KUKA KRL program: MyProgram_115().src

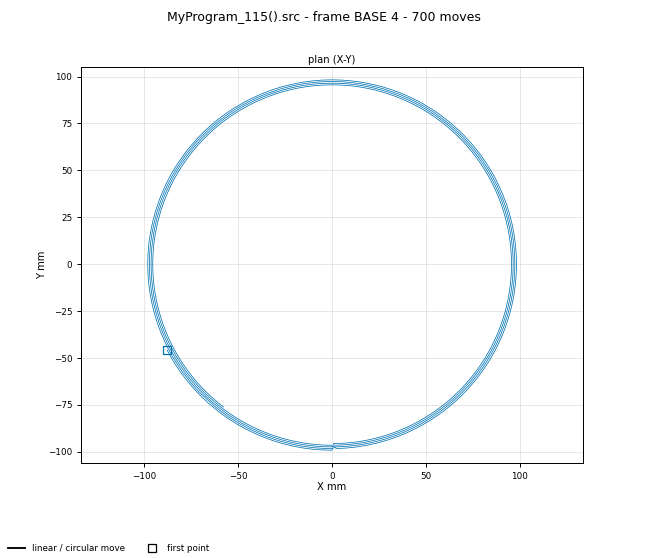
[picture p0: tool path of MyProgram_115().src in frame BASE 4, 700 of 700 moves have a stored position in this frame; points joined in program order, loops and branches not executed]
&ACCESS RVP
&REL 1
&PARAM TEMPLATE = C:\KRC\Roboter\Template\vorgabe
&PARAM EDITMASK = *
DEF MyProgram_115()
; ---- Setting reference (Base) ----
$BASE = BASE_DATA[4]

; --------------------------
; ---- Setting tool (TCP) ----
$TOOL = TOOL_DATA[3]
; --------------------------

$VEL.CP = VEL_APROX_PRINT
Startdeposition()
$VEL.CP = VEL_PRINT
LIN {X -87.9796,Y -45.6346,Z 99,A -156.4793,B 24.9343,C -1.8721,E1 24.8586,E2 241.8644} C_DIS
LIN {X -86.3816,Y -48.5897,Z 99,A -154.8089,B 24.9353,C -1.8576,E1 24.8608,E2 240.2197} C_DIS
LIN {X -84.702,Y -51.4607,Z 99,A -152.4572,B 24.9346,C -1.8672,E1 24.8642,E2 237.8331} C_DIS
LIN {X -82.3707,Y -55.1181,Z 99,A -150.0558,B 24.9354,C -1.8571,E1 24.8679,E2 235.4438} C_DIS
LIN {X -80.7403,Y -57.4774,Z 99,A -147.4324,B 24.9333,C -1.8865,E1 24.8723,E2 232.7375} C_DIS
LIN {X -77.3944,Y -61.9119,Z 99,A -145.2941,B 24.9364,C -1.8414,E1 24.8758,E2 230.6966} C_DIS
LIN {X -72.9328,Y -67.1078,Z 99,A -141.2258,B 24.9368,C -1.8361,E1 24.8833,E2 226.6225} C_DIS
LIN {X -70.3897,Y -69.7707,Z 99,A -138.1583,B 24.9348,C -1.8645,E1 24.8895,E2 223.4743} C_DIS
LIN {X -66.5722,Y -73.4243,Z 99,A -135.9548,B 24.9373,C -1.8283,E1 24.8938,E2 221.3481} C_DIS
LIN {X -64.5573,Y -75.2007,Z 99,A -133.5935,B 24.9356,C -1.8539,E1 24.899,E2 218.9168} C_DIS
LIN {X -60.7037,Y -78.3439,Z 99,A -131.5906,B 24.9381,C -1.8177,E1 24.9032,E2 216.9924} C_DIS
LIN {X -57.0304,Y -81.0586,Z 99,A -129.0585,B 24.9386,C -1.8094,E1 24.9089,E2 214.4714} C_DIS
LIN {X -53.8485,Y -83.2053,Z 99,A -126.6505,B 24.9384,C -1.8125,E1 24.9145,E2 212.0479} C_DIS
LIN {X -50.892,Y -85.0464,Z 99,A -124.5261,B 24.9384,C -1.8135,E1 24.9196,E2 209.9146} C_DIS
LIN {X -47.2587,Y -87.1163,Z 99,A -122.248,B 24.9389,C -1.8053,E1 24.9252,E2 207.6496} C_DIS
LIN {X -44.1537,Y -88.7306,Z 99,A -120.2492,B 24.9391,C -1.8018,E1 24.9301,E2 205.6535} C_DIS
LIN {X -40.0948,Y -90.6385,Z 99,A -117.5727,B 24.9391,C -1.8018,E1 24.9369,E2 202.9703} C_DIS
LIN {X -36.8273,Y -92.0148,Z 99,A -115.7096,B 24.9397,C -1.7931,E1 24.9417,E2 201.1239} C_DIS
LIN {X -32.0757,Y -93.7762,Z 99,A -112.6664,B 24.9397,C -1.7946,E1 24.9497,E2 198.0711} C_DIS
LIN {X -29.2016,Y -94.7097,Z 99,A -111.0211,B 24.94,C -1.7896,E1 24.9541,E2 196.4347} C_DIS
LIN {X -26.1849,Y -95.5883,Z 99,A -108.5473,B 24.9384,C -1.8125,E1 24.9609,E2 193.9027} C_DIS
LIN {X -22.6221,Y -96.4935,Z 99,A -106.9162,B 24.9397,C -1.7932,E1 24.9652,E2 192.3152} C_DIS
LIN {X -18.9638,Y -97.2783,Z 99,A -104.6871,B 24.9397,C -1.7947,E1 24.9713,E2 190.0799} C_DIS
LIN {X -15.5993,Y -97.875,Z 99,A -102.0723,B 24.9381,C -1.8179,E1 24.9787,E2 187.4077} C_DIS
LIN {X -11.2084,Y -98.4739,Z 99,A -100.3885,B 24.9403,C -1.7848,E1 24.9832,E2 185.8012} C_DIS
LIN {X -7.2101,Y -98.847,Z 99,A -97.791,B 24.9396,C -1.7949,E1 24.9904,E2 183.1785} C_DIS
LIN {X -0.3589,Y -99.1089,Z 99,A -93.8886,B 24.9397,C -1.7932,E1 25.0013,E2 179.2797} C_DIS
LIN {X -0.3589,Y -99.1089,Z 99,A -93.8886,B 24.9397,C -1.7932,E1 25.0013,E2 179.2797} C_DIS
Enddeposition()
LIN {X 0.6693,Y -98.2189,Z 99,A -93.8289,B 24.94,C -1.7889,E1 25.0015,E2 179.2303} C_DIS
Startdeposition()
$VEL.CP = VEL_PRINT
LIN {X -4.2372,Y -98.1313,Z 99,A -96.6951,B 24.94,C -1.7882,E1 24.9935,E2 182.0983} C_DIS
LIN {X -8.8121,Y -97.8269,Z 99,A -99.6848,B 24.9408,C -1.7766,E1 24.9851,E2 185.1165} C_DIS
LIN {X -11.6628,Y -97.5282,Z 99,A -101.9207,B 24.9422,C -1.7566,E1 24.9787,E2 187.4014} C_DIS
LIN {X -14.8528,Y -97.0934,Z 99,A -103.5542,B 24.9416,C -1.7658,E1 24.9742,E2 189.0145} C_DIS
LIN {X -17.6713,Y -96.6205,Z 99,A -105.1253,B 24.9413,C -1.7698,E1 24.97,E2 190.5777} C_DIS
LIN {X -21.247,Y -95.8977,Z 99,A -107.2347,B 24.9412,C -1.7714,E1 24.9642,E2 192.6858} C_DIS
LIN {X -27.1234,Y -94.4042,Z 99,A -110.6543,B 24.9408,C -1.7776,E1 24.955,E2 196.0956} C_DIS
LIN {X -30.1752,Y -93.4728,Z 99,A -112.5555,B 24.9408,C -1.7776,E1 24.9499,E2 198.0002} C_DIS
LIN {X -35.0219,Y -91.7671,Z 99,A -115.6071,B 24.9408,C -1.7783,E1 24.9419,E2 201.0563} C_DIS
LIN {X -37.3216,Y -90.8565,Z 99,A -117.2902,B 24.9412,C -1.7714,E1 24.9375,E2 202.7597} C_DIS
LIN {X -42.4401,Y -88.5808,Z 99,A -119.9202,B 24.9395,C -1.7973,E1 24.9309,E2 205.3344} C_DIS
LIN {X -44.6777,Y -87.4735,Z 99,A -121.7115,B 24.9401,C -1.7874,E1 24.9264,E2 207.154} C_DIS
LIN {X -47.4006,Y -86.0303,Z 99,A -123.6442,B 24.9403,C -1.7851,E1 24.9216,E2 209.0977} C_DIS
LIN {X -50.7015,Y -84.1261,Z 99,A -125.8121,B 24.9399,C -1.7902,E1 24.9164,E2 211.26} C_DIS
LIN {X -52.833,Y -82.8037,Z 99,A -127.3649,B 24.9399,C -1.7894,E1 24.9127,E2 212.8197} C_DIS
LIN {X -55.9629,Y -80.721,Z 99,A -129.7908,B 24.9403,C -1.785,E1 24.9071,E2 215.2643} C_DIS
LIN {X -59.7569,Y -77.9544,Z 99,A -132.7771,B 24.9405,C -1.7814,E1 24.9004,E2 218.2698} C_DIS
LIN {X -62.6614,Y -75.6391,Z 99,A -134.7841,B 24.9399,C -1.7908,E1 24.8961,E2 220.2619} C_DIS
LIN {X -70.1603,Y -68.7416,Z 99,A -140.19,B 24.9378,C -1.8212,E1 24.8852,E2 225.6178} C_DIS
LIN {X -71.8208,Y -67.0047,Z 99,A -142.6978,B 24.9401,C -1.7872,E1 24.8803,E2 228.2174} C_DIS
LIN {X -75.1999,Y -63.1899,Z 99,A -144.6057,B 24.9373,C -1.8295,E1 24.877,E2 230.0332} C_DIS
LIN {X -79.9184,Y -57.1031,Z 99,A -149.1944,B 24.9367,C -1.8372,E1 24.8692,E2 234.6255} C_DIS
LIN {X -81.4693,Y -54.8681,Z 99,A -151.0136,B 24.937,C -1.8335,E1 24.8663,E2 236.4626} C_DIS
LIN {X -84.5611,Y -49.9712,Z 99,A -154.2394,B 24.936,C -1.8474,E1 24.8616,E2 239.6718} C_DIS
LIN {X -86.4889,Y -46.5562,Z 99,A -156.7026,B 24.936,C -1.8477,E1 24.8582,E2 242.1471} C_DIS
LIN {X -88.1614,Y -43.3058,Z 99,A -158.6261,B 24.9351,C -1.8605,E1 24.8558,E2 244.0503} C_DIS
LIN {X -89.5289,Y -40.4016,Z 99,A -160.5798,B 24.9349,C -1.8632,E1 24.8535,E2 246.0084} C_DIS
LIN {X -91.4852,Y -35.7517,Z 99,A -163.3808,B 24.934,C -1.8763,E1 24.8506,E2 248.7936} C_DIS
LIN {X -92.4618,Y -33.1485,Z 99,A -165.732,B 24.9353,C -1.8572,E1 24.8483,E2 251.2037} C_DIS
LIN {X -93.5984,Y -29.784,Z 99,A -167.1976,B 24.9335,C -1.8832,E1 24.8471,E2 252.6157} C_DIS
LIN {X -94.6082,Y -26.4034,Z 99,A -169.3529,B 24.9333,C -1.8862,E1 24.8454,E2 254.7762} C_DIS
LIN {X -95.2785,Y -23.876,Z 99,A -170.9762,B 24.9333,C -1.8877,E1 24.8442,E2 256.4055} C_DIS
LIN {X -96.0802,Y -20.4103,Z 99,A -173.0544,B 24.9328,C -1.894,E1 24.843,E2 258.481} C_DIS
LIN {X -96.7044,Y -17.2045,Z 99,A -174.9863,B 24.9324,C -1.8991,E1 24.842,E2 260.4121} C_DIS
LIN {X -97.2841,Y -13.5493,Z 99,A -176.9634,B 24.9315,C -1.9118,E1 24.8412,E2 262.3707} C_DIS
LIN {X -97.6646,Y -10.4583,Z 99,A -178.9019,B 24.9314,C -1.9136,E1 24.8406,E2 264.3165} C_DIS
LIN {X -97.9778,Y -6.9396,Z 99,A 178.9434,B 24.9311,C -1.9171,E1 24.8401,E2 266.4758} C_DIS
LIN {X -98.1766,Y -3.0096,Z 99,A 176.7382,B 24.9304,C -1.9274,E1 24.8398,E2 268.6697} C_DIS
LIN {X -98.2194,Y 0.859,Z 99,A 174.7208,B 24.9293,C -1.9424,E1 24.8398,E2 270.6634} C_DIS
LIN {X -98.1684,Y 3.2759,Z 99,A 173.0765,B 24.9295,C -1.9394,E1 24.8399,E2 272.3249} C_DIS
LIN {X -98.0007,Y 6.6012,Z 99,A 170.3743,B 24.9308,C -1.9212,E1 24.8404,E2 275.0868} C_DIS
LIN {X -97.623,Y 10.8528,Z 99,A 168.69,B 24.9283,C -1.9551,E1 24.8409,E2 276.7004} C_DIS
LIN {X -97.2609,Y 13.7126,Z 99,A 166.8511,B 24.9283,C -1.9554,E1 24.8416,E2 278.5495} C_DIS
LIN {X -96.2313,Y 19.6787,Z 99,A 163.3352,B 24.9274,C -1.9672,E1 24.8433,E2 282.058} C_DIS
LIN {X -95.4672,Y 23.1029,Z 99,A 160.3611,B 24.9292,C -1.9439,E1 24.8453,E2 285.1052} C_DIS
LIN {X -94.1956,Y 27.8372,Z 99,A 158.004,B 24.9273,C -1.9689,E1 24.8471,E2 287.416} C_DIS
LIN {X -92.5031,Y 33.0331,Z 99,A 155.2903,B 24.9254,C -1.9942,E1 24.8495,E2 290.0851} C_DIS
LIN {X -91.607,Y 35.4417,Z 99,A 153.1393,B 24.9267,C -1.9777,E1 24.8517,E2 292.2874} C_DIS
LIN {X -90.2742,Y 38.7115,Z 99,A 151.0056,B 24.9264,C -1.9816,E1 24.854,E2 294.4238} C_DIS
LIN {X -88.7429,Y 42.1028,Z 99,A 149.5708,B 24.9241,C -2.0119,E1 24.8556,E2 295.794} C_DIS
LIN {X -87.6054,Y 44.4197,Z 99,A 147.8824,B 24.9242,C -2.0104,E1 24.8578,E2 297.495} C_DIS
LIN {X -85.5205,Y 48.3133,Z 99,A 145.4516,B 24.9233,C -2.0227,E1 24.861,E2 299.9094} C_DIS
LIN {X -83.4828,Y 51.7536,Z 99,A 142.425,B 24.9245,C -2.0067,E1 24.8654,E2 302.9896} C_DIS
LIN {X -81.5716,Y 54.7167,Z 99,A 140.6129,B 24.9235,C -2.0204,E1 24.8682,E2 304.7782} C_DIS
LIN {X -78.2992,Y 59.3051,Z 99,A 137.7295,B 24.9218,C -2.0426,E1 24.8729,E2 307.6227} C_DIS
LIN {X -75.9566,Y 62.277,Z 99,A 135,B 24.9226,C -2.0312,E1 24.8777,E2 310.3919} C_DIS
LIN {X -70.7131,Y 68.1716,Z 99,A 130.8132,B 24.9207,C -2.0565,E1 24.8855,E2 314.5371} C_DIS
LIN {X -67.7866,Y 71.0819,Z 99,A 128.1614,B 24.9209,C -2.0542,E1 24.8908,E2 317.2056} C_DIS
LIN {X -64.3882,Y 74.1752,Z 99,A 125.2789,B 24.9209,C -2.0536,E1 24.8969,E2 320.1009} C_DIS
LIN {X -61.2392,Y 76.7962,Z 99,A 122.5585,B 24.9214,C -2.0478,E1 24.9029,E2 322.8451} C_DIS
LIN {X -58.1125,Y 79.1875,Z 99,A 121.0253,B 24.919,C -2.078,E1 24.9061,E2 324.312} C_DIS
LIN {X -55.5869,Y 80.9823,Z 99,A 119.1347,B 24.919,C -2.0788,E1 24.9105,E2 326.2072} C_DIS
LIN {X -53.0483,Y 82.6655,Z 99,A 117.3096,B 24.9188,C -2.0806,E1 24.9147,E2 328.0339} C_DIS
LIN {X -46.7576,Y 86.3796,Z 99,A 112.9813,B 24.9184,C -2.0859,E1 24.9252,E2 332.3625} C_DIS
LIN {X -43.5021,Y 88.0641,Z 99,A 110.8049,B 24.9182,C -2.0881,E1 24.9306,E2 334.5396} C_DIS
LIN {X -37.4457,Y 90.806,Z 99,A 106.9454,B 24.9177,C -2.0944,E1 24.9405,E2 338.3932} C_DIS
LIN {X -34.403,Y 92.0017,Z 99,A 104.5204,B 24.9189,C -2.0793,E1 24.9469,E2 340.8592} C_DIS
LIN {X -30.9828,Y 93.2092,Z 99,A 102.7552,B 24.9178,C -2.0938,E1 24.9515,E2 342.5932} C_DIS
LIN {X -27.1596,Y 94.394,Z 99,A 100.5654,B 24.9172,C -2.1014,E1 24.9573,E2 344.7687} C_DIS
LIN {X -23.8098,Y 95.2948,Z 99,A 98.4109,B 24.9174,C -2.0989,E1 24.9632,E2 346.9323} C_DIS
LIN {X -18.4947,Y 96.4658,Z 99,A 95.5222,B 24.9164,C -2.1116,E1 24.971,E2 349.7944} C_DIS
LIN {X -15.6439,Y 96.9706,Z 99,A 93.6883,B 24.9167,C -2.1077,E1 24.976,E2 351.6393} C_DIS
LIN {X -11.0151,Y 97.6039,Z 99,A 90.8548,B 24.9169,C -2.1056,E1 24.9839,E2 354.4798} C_DIS
LIN {X -6.5203,Y 98.0061,Z 99,A 88.4661,B 24.9161,C -2.1153,E1 24.9905,E2 356.8464} C_DIS
LIN {X -3.7024,Y 98.1543,Z 99,A 85.9121,B 24.9186,C -2.084,E1 24.9979,E2 359.4752} C_DIS
LIN {X 0.739,Y 98.22,Z 99,A 84.3272,B 24.9157,C -2.12,E1 25.002,E2 360.9748} C_DIS
LIN {X 5.0113,Y 98.0957,Z 99,A 81.8155,B 24.9157,C -2.1195,E1 25.0091,E2 363.487} C_DIS
LIN {X 9.2561,Y 97.7859,Z 99,A 78.8188,B 24.9172,C -2.101,E1 25.0175,E2 366.526} C_DIS
LIN {X 14.5628,Y 97.1382,Z 99,A 75.9511,B 24.9166,C -2.1092,E1 25.0254,E2 369.3718} C_DIS
LIN {X 17.9733,Y 96.5661,Z 99,A 73.8851,B 24.9168,C -2.1067,E1 25.0311,E2 371.4416} C_DIS
LIN {X 24.0268,Y 95.2397,Z 99,A 70.4453,B 24.9164,C -2.1112,E1 25.0404,E2 374.866} C_DIS
LIN {X 26.8049,Y 94.4945,Z 99,A 68.7342,B 24.9166,C -2.1089,E1 25.045,E2 376.5798} C_DIS
LIN {X 31.2762,Y 93.1102,Z 99,A 65.7465,B 24.9175,C -2.0973,E1 25.053,E2 379.5893} C_DIS
LIN {X 35.2372,Y 91.6857,Z 99,A 63.1236,B 24.9182,C -2.0889,E1 25.0599,E2 382.2266} C_DIS
LIN {X 39.7787,Y 89.8092,Z 99,A 60.5994,B 24.9174,C -2.0983,E1 25.0663,E2 384.7225} C_DIS
LIN {X 42.5653,Y 88.5206,Z 99,A 58.8919,B 24.9174,C -2.0993,E1 25.0706,E2 386.4234} C_DIS
LIN {X 45.7119,Y 86.9375,Z 99,A 56.2233,B 24.9193,C -2.074,E1 25.0773,E2 389.1444} C_DIS
LIN {X 49.1089,Y 85.065,Z 99,A 54.6522,B 24.9176,C -2.0963,E1 25.081,E2 390.6579} C_DIS
LIN {X 52.9984,Y 82.6975,Z 99,A 51.6171,B 24.919,C -2.0782,E1 25.0883,E2 393.7263} C_DIS
LIN {X 56.5537,Y 80.3103,Z 99,A 49.1582,B 24.9192,C -2.0754,E1 25.0939,E2 396.1833} C_DIS
LIN {X 61.5521,Y 76.5453,Z 99,A 45.9308,B 24.9185,C -2.0847,E1 25.101,E2 399.3768} C_DIS
LIN {X 63.6975,Y 74.7685,Z 99,A 43.4325,B 24.9213,C -2.0488,E1 25.1065,E2 401.9504} C_DIS
LIN {X 67.0136,Y 71.8125,Z 99,A 41.8291,B 24.9188,C -2.0808,E1 25.1096,E2 403.4718} C_DIS
LIN {X 70.2791,Y 68.6213,Z 99,A 38.0175,B 24.9226,C -2.0317,E1 25.1173,E2 407.3831} C_DIS
LIN {X 73.7212,Y 64.908,Z 99,A 36.2315,B 24.9197,C -2.0693,E1 25.1205,E2 409.0724} C_DIS
LIN {X 75.4284,Y 62.915,Z 99,A 34.3583,B 24.921,C -2.0526,E1 25.1239,E2 410.9764} C_DIS
LIN {X 77.4398,Y 60.4247,Z 99,A 32.5137,B 24.9213,C -2.0489,E1 25.1271,E2 412.8211} C_DIS
LIN {X 79.6298,Y 57.5076,Z 99,A 29.9603,B 24.9229,C -2.0274,E1 25.1314,E2 415.413} C_DIS
LIN {X 81.7209,Y 54.4946,Z 99,A 27.7548,B 24.9235,C -2.0194,E1 25.1348,E2 417.6264} C_DIS
LIN {X 83.8285,Y 51.1911,Z 99,A 26.1333,B 24.922,C -2.0389,E1 25.1371,E2 419.1936} C_DIS
LIN {X 85.3464,Y 48.6193,Z 99,A 24.2068,B 24.9229,C -2.0271,E1 25.1398,E2 421.138} C_DIS
LIN {X 87.3551,Y 44.9093,Z 99,A 21.9087,B 24.9229,C -2.0266,E1 25.1428,E2 423.4251} C_DIS
LIN {X 89.3446,Y 40.8104,Z 99,A 18.667,B 24.9253,C -1.9966,E1 25.1467,E2 426.7204} C_DIS
LIN {X 90.8949,Y 37.2273,Z 99,A 16.931,B 24.9242,C -2.0109,E1 25.1485,E2 428.4129} C_DIS
LIN {X 92.6114,Y 32.7238,Z 99,A 14.1219,B 24.9248,C -2.0027,E1 25.1512,E2 431.2256} C_DIS
LIN {X 93.5223,Y 30.0221,Z 99,A 12.5231,B 24.925,C -2.0002,E1 25.1526,E2 432.8212} C_DIS
LIN {X 94.5572,Y 26.5834,Z 99,A 10.5146,B 24.9252,C -1.9973,E1 25.1542,E2 434.8252} C_DIS
LIN {X 95.7288,Y 21.9936,Z 99,A 8.0802,B 24.9249,C -2.0017,E1 25.1558,E2 437.2352} C_DIS
LIN {X 96.2495,Y 19.59,Z 99,A 6.3366,B 24.9261,C -1.9851,E1 25.1568,E2 439.0078} C_DIS
LIN {X 97.0337,Y 15.2384,Z 99,A 3.3697,B 24.9278,C -1.9618,E1 25.1582,E2 442.0122} C_DIS
LIN {X 97.6877,Y 10.2376,Z 99,A 0.8517,B 24.9273,C -1.9691,E1 25.159,E2 444.4982} C_DIS
LIN {X 98.1268,Y 4.3414,Z 99,A -2.2125,B 24.927,C -1.9732,E1 25.1597,E2 447.5344} C_DIS
LIN {X 98.204,Y -1.9222,Z 99,A -5.7141,B 24.9274,C -1.9674,E1 25.1597,E2 451.0289} C_DIS
LIN {X 97.9726,Y -7.0165,Z 99,A -9.4841,B 24.9304,C -1.9264,E1 25.1592,E2 454.8733} C_DIS
LIN {X 97.5536,Y -11.4457,Z 99,A -11.7511,B 24.9301,C -1.9309,E1 25.1585,E2 457.1161} C_DIS
LIN {X 97.0799,Y -14.9401,Z 99,A -14.3987,B 24.9322,C -1.9011,E1 25.1574,E2 459.8184} C_DIS
LIN {X 96.4009,Y -18.832,Z 99,A -15.8277,B 24.9303,C -1.9281,E1 25.1567,E2 461.1754} C_DIS
LIN {X 95.5332,Y -22.8327,Z 99,A -18.4033,B 24.9314,C -1.9131,E1 25.1552,E2 463.7716} C_DIS
LIN {X 94.7265,Y -25.9755,Z 99,A -20.7733,B 24.9332,C -1.8883,E1 25.1534,E2 466.1863} C_DIS
LIN {X 93.8078,Y -29.117,Z 99,A -21.7976,B 24.9311,C -1.9171,E1 25.1527,E2 467.1367} C_DIS
LIN {X 92.2233,Y -33.8024,Z 99,A -24.9868,B 24.9326,C -1.8961,E1 25.1498,E2 470.3577} C_DIS
LIN {X 91.2153,Y -36.4388,Z 99,A -26.8626,B 24.9336,C -1.882,E1 25.1478,E2 472.2564} C_DIS
LIN {X 89.7318,Y -39.9512,Z 99,A -28.9823,B 24.9338,C -1.8793,E1 25.1454,E2 474.3708} C_DIS
LIN {X 88.2705,Y -43.0857,Z 99,A -31.4641,B 24.9355,C -1.8551,E1 25.1424,E2 476.8964} C_DIS
LIN {X 86.6504,Y -46.2556,Z 99,A -32.8541,B 24.934,C -1.8758,E1 25.1407,E2 478.2302} C_DIS
LIN {X 84.7613,Y -49.6312,Z 99,A -35.3481,B 24.9352,C -1.8599,E1 25.1372,E2 480.7487} C_DIS
LIN {X 82.971,Y -52.5724,Z 99,A -38.1757,B 24.9377,C -1.8224,E1 25.1328,E2 483.6505} C_DIS
LIN {X 80.1308,Y -56.8053,Z 99,A -40.6335,B 24.9369,C -1.8341,E1 25.129,E2 486.0687} C_DIS
LIN {X 78.1599,Y -59.4894,Z 99,A -41.9721,B 24.9357,C -1.8523,E1 25.1268,E2 487.358} C_DIS
LIN {X 76.5852,Y -61.5029,Z 99,A -43.6658,B 24.9365,C -1.8404,E1 25.1238,E2 489.0719} C_DIS
LIN {X 74.2917,Y -64.2548,Z 99,A -45.7261,B 24.9368,C -1.8361,E1 25.1201,E2 491.1329} C_DIS
LIN {X 72.0089,Y -66.8035,Z 99,A -47.7759,B 24.9373,C -1.829,E1 25.1162,E2 493.1906} C_DIS
LIN {X 69.4466,Y -69.4638,Z 99,A -49.9069,B 24.9376,C -1.8246,E1 25.112,E2 495.3228} C_DIS
LIN {X 66.9301,Y -71.891,Z 99,A -51.9343,B 24.9379,C -1.8202,E1 25.1079,E2 497.3521} C_DIS
LIN {X 64.2959,Y -74.2557,Z 99,A -53.986,B 24.9382,C -1.816,E1 25.1036,E2 499.4058} C_DIS
LIN {X 61.5657,Y -76.5343,Z 99,A -56.0026,B 24.9383,C -1.8136,E1 25.0993,E2 501.4203} C_DIS
LIN {X 58.8534,Y -78.6385,Z 99,A -57.8721,B 24.9383,C -1.8144,E1 25.0951,E2 503.281} C_DIS
LIN {X 56.3775,Y -80.4313,Z 99,A -60.5491,B 24.9408,C -1.7768,E1 25.0889,E2 506.0377} C_DIS
LIN {X 52.4164,Y -83.0688,Z 99,A -62.2949,B 24.9386,C -1.8105,E1 25.085,E2 507.6982} C_DIS
LIN {X 48.4774,Y -85.4265,Z 99,A -65.0774,B 24.9392,C -1.8016,E1 25.0782,E2 510.4933} C_DIS
LIN {X 45.2759,Y -87.1671,Z 99,A -67.2226,B 24.9395,C -1.7971,E1 25.0729,E2 512.6428} C_DIS
LIN {X 42.5313,Y -88.537,Z 99,A -69.0261,B 24.9397,C -1.7937,E1 25.0684,E2 514.4496} C_DIS
LIN {X 39.6623,Y -89.8599,Z 99,A -70.9486,B 24.9401,C -1.7879,E1 25.0635,E2 516.3811} C_DIS
LIN {X 36.0867,Y -91.3537,Z 99,A -73.4145,B 24.9408,C -1.7769,E1 25.0571,E2 518.8673} C_DIS
LIN {X 32.52,Y -92.6831,Z 99,A -75.3654,B 24.9403,C -1.7841,E1 25.052,E2 520.7971} C_DIS
LIN {X 29.2556,Y -93.7648,Z 99,A -77.142,B 24.9399,C -1.7903,E1 25.0473,E2 522.5558} C_DIS
LIN {X 26.5194,Y -94.5753,Z 99,A -79.1248,B 24.9408,C -1.7765,E1 25.0419,E2 524.5678} C_DIS
LIN {X 23.0106,Y -95.4898,Z 99,A -81.6817,B 24.9421,C -1.7581,E1 25.0349,E2 527.1647} C_DIS
LIN {X 19.4296,Y -96.2824,Z 99,A -83.0743,B 24.9404,C -1.7838,E1 25.0312,E2 528.4946} C_DIS
LIN {X 14.2618,Y -97.1829,Z 99,A -86.1327,B 24.9405,C -1.7815,E1 25.0228,E2 531.5553} C_DIS
LIN {X 11.5148,Y -97.5455,Z 99,A -88.643,B 24.9428,C -1.7477,E1 25.0156,E2 534.1437} C_DIS
LIN {X 7.2682,Y -97.954,Z 99,A -90.2392,B 24.9407,C -1.7791,E1 25.0114,E2 535.6648} C_DIS
LIN {X 2.4421,Y -98.194,Z 99,A -93.1283,B 24.9409,C -1.7754,E1 25.0033,E2 538.5618} C_DIS
LIN {X 2.4421,Y -98.194,Z 99,A -93.1283,B 24.9409,C -1.7754,E1 25.0033,E2 538.5618} C_DIS
Enddeposition()
LIN {X 0.6795,Y -97.3292,Z 99,A -94.8368,B 24.9415,C -1.7664,E1 24.9985,E2 540.2915} C_DIS
Startdeposition()
$VEL.CP = VEL_PRINT
LIN {X 2.7609,Y -97.2973,Z 99,A -92.3696,B 24.9385,C -1.8114,E1 25.0057,E2 537.7178} C_DIS
LIN {X 6.1522,Y -97.1425,Z 99,A -90.0447,B 24.9376,C -1.8242,E1 25.0122,E2 535.3633} C_DIS
LIN {X 11.274,Y -96.6811,Z 99,A -87.1052,B 24.9377,C -1.8227,E1 25.0204,E2 532.4294} C_DIS
LIN {X 14.8657,Y -96.1943,Z 99,A -85.2733,B 24.9384,C -1.813,E1 25.0254,E2 530.6221} C_DIS
LIN {X 18.8901,Y -95.4869,Z 99,A -82.7672,B 24.938,C -1.8186,E1 25.0323,E2 528.1055} C_DIS
LIN {X 22.4498,Y -94.7135,Z 99,A -80.5208,B 24.9376,C -1.8244,E1 25.0385,E2 525.8484} C_DIS
LIN {X 25.749,Y -93.8694,Z 99,A -78.4867,B 24.9374,C -1.8276,E1 25.044,E2 523.8098} C_DIS
LIN {X 29.2145,Y -92.8494,Z 99,A -76.1919,B 24.9368,C -1.8364,E1 25.0501,E2 521.4982} C_DIS
LIN {X 33.2362,Y -91.4861,Z 99,A -73.2488,B 24.9354,C -1.8566,E1 25.058,E2 518.5135} C_DIS
LIN {X 37.0035,Y -90.0288,Z 99,A -71.6188,B 24.9371,C -1.8315,E1 25.062,E2 516.9466} C_DIS
LIN {X 39.6241,Y -88.9069,Z 99,A -69.8166,B 24.9366,C -1.8387,E1 25.0667,E2 515.1317} C_DIS
LIN {X 42.3266,Y -87.6518,Z 99,A -68.1387,B 24.9366,C -1.8386,E1 25.0709,E2 513.4584} C_DIS
LIN {X 45.5815,Y -86.0043,Z 99,A -66.213,B 24.937,C -1.8337,E1 25.0756,E2 511.5494} C_DIS
LIN {X 47.519,Y -84.9488,Z 99,A -64.0147,B 24.9344,C -1.8706,E1 25.0812,E2 509.2705} C_DIS
LIN {X 51.0825,Y -82.8568,Z 99,A -61.6838,B 24.9344,C -1.8712,E1 25.0867,E2 506.9455} C_DIS
LIN {X 54.0996,Y -80.9163,Z 99,A -59.831,B 24.9348,C -1.8654,E1 25.091,E2 505.1127} C_DIS
LIN {X 58.6732,Y -77.6651,Z 99,A -56.7781,B 24.935,C -1.8625,E1 25.0978,E2 502.0773} C_DIS
LIN {X 61.5832,Y -75.379,Z 99,A -54.6217,B 24.9347,C -1.8665,E1 25.1025,E2 499.9197} C_DIS
LIN {X 64.2602,Y -73.1099,Z 99,A -52.5485,B 24.9343,C -1.8715,E1 25.1069,E2 497.8428} C_DIS
LIN {X 67.0011,Y -70.6072,Z 99,A -50.4221,B 24.9341,C -1.8744,E1 25.1112,E2 495.7183} C_DIS
LIN {X 69.2046,Y -68.4476,Z 99,A -48.6255,B 24.9339,C -1.878,E1 25.1148,E2 493.9205} C_DIS
LIN {X 71.6573,Y -65.8755,Z 99,A -46.581,B 24.9336,C -1.8814,E1 25.1187,E2 491.877} C_DIS
LIN {X 74.019,Y -63.2102,Z 99,A -44.4945,B 24.9333,C -1.8864,E1 25.1225,E2 489.788} C_DIS
LIN {X 76.2827,Y -60.4592,Z 99,A -42.4736,B 24.9331,C -1.889,E1 25.1261,E2 487.7705} C_DIS
LIN {X 79.5834,Y -56.0462,Z 99,A -38.3599,B 24.93,C -1.9322,E1 25.1329,E2 483.5747} C_DIS
LIN {X 82.155,Y -52.2024,Z 99,A -36.3882,B 24.9316,C -1.9102,E1 25.1358,E2 481.6649} C_DIS
LIN {X 85.1566,Y -47.1468,Z 99,A -32.8353,B 24.9306,C -1.9238,E1 25.1408,E2 478.0982} C_DIS
LIN {X 87.494,Y -42.6551,Z 99,A -29.9743,B 24.9303,C -1.9279,E1 25.1444,E2 475.2427} C_DIS
LIN {X 88.9843,Y -39.4523,Z 99,A -27.8809,B 24.9298,C -1.9348,E1 25.1468,E2 473.1445} C_DIS
LIN {X 90.2419,Y -36.48,Z 99,A -26.0268,B 24.9295,C -1.9388,E1 25.1488,E2 471.2911} C_DIS
LIN {X 91.3472,Y -33.6171,Z 99,A -23.9892,B 24.9284,C -1.9536,E1 25.1508,E2 469.23} C_DIS
LIN {X 93.1093,Y -28.3764,Z 99,A -20.8704,B 24.9281,C -1.9584,E1 25.1535,E2 466.1177} C_DIS
LIN {X 94.1676,Y -24.637,Z 99,A -18.791,B 24.9281,C -1.9573,E1 25.155,E2 464.0526} C_DIS
LIN {X 94.7908,Y -22.1155,Z 99,A -17.0726,B 24.9273,C -1.9697,E1 25.1561,E2 462.3149} C_DIS
LIN {X 95.5103,Y -18.7688,Z 99,A -14.9623,B 24.9265,C -1.98,E1 25.1573,E2 460.1928} C_DIS
LIN {X 96.2935,Y -14.2191,Z 99,A -12.5621,B 24.9268,C -1.9761,E1 25.1583,E2 457.8159} C_DIS
LIN {X 96.6677,Y -11.3886,Z 99,A -10.9582,B 24.9266,C -1.9785,E1 25.1588,E2 456.2157} C_DIS
LIN {X 96.9696,Y -8.4551,Z 99,A -9.0924,B 24.9258,C -1.9892,E1 25.1593,E2 454.3358} C_DIS
LIN {X 97.2753,Y -3.4781,Z 99,A -6.2139,B 24.9253,C -1.9964,E1 25.1597,E2 451.4573} C_DIS
LIN {X 97.3347,Y -0.5369,Z 99,A -4.0288,B 24.9235,C -2.0201,E1 25.1597,E2 449.2294} C_DIS
LIN {X 97.2865,Y 3.112,Z 99,A -2.45,B 24.9247,C -2.0043,E1 25.1597,E2 447.6972} C_DIS
LIN {X 97.0318,Y 7.6924,Z 99,A 0.2957,B 24.9239,C -2.0147,E1 25.1592,E2 444.9432} C_DIS
LIN {X 96.6465,Y 11.5698,Z 99,A 2.4563,B 24.9237,C -2.0168,E1 25.1585,E2 442.7906} C_DIS
LIN {X 96.1397,Y 15.2189,Z 99,A 4.8764,B 24.9225,C -2.0335,E1 25.1575,E2 440.3451} C_DIS
LIN {X 95.3723,Y 19.4544,Z 99,A 7.1675,B 24.9225,C -2.0319,E1 25.1563,E2 438.0714} C_DIS
LIN {X 94.7055,Y 22.4848,Z 99,A 9.282,B 24.9213,C -2.0489,E1 25.155,E2 435.9291} C_DIS
LIN {X 93.6368,Y 26.5799,Z 99,A 11.4571,B 24.9217,C -2.044,E1 25.1534,E2 433.7778} C_DIS
LIN {X 92.4495,Y 30.4582,Z 99,A 14.6632,B 24.9186,C -2.0835,E1 25.1506,E2 430.4968} C_DIS
LIN {X 90.9071,Y 34.7902,Z 99,A 16.5146,B 24.9206,C -2.0577,E1 25.1488,E2 428.7165} C_DIS
LIN {X 88.3231,Y 40.9074,Z 99,A 20.4688,B 24.9196,C -2.0706,E1 25.1444,E2 424.7534} C_DIS
LIN {X 86.88,Y 43.891,Z 99,A 22.3993,B 24.9192,C -2.0753,E1 25.142,E2 422.8223} C_DIS
LIN {X 85.2962,Y 46.8957,Z 99,A 24.4809,B 24.9186,C -2.0839,E1 25.1392,E2 420.7312} C_DIS
LIN {X 83.3931,Y 50.2007,Z 99,A 26.9403,B 24.9174,C -2.0983,E1 25.1357,E2 418.2505} C_DIS
LIN {X 80.9671,Y 54.0273,Z 99,A 29.1173,B 24.9184,C -2.0861,E1 25.1325,E2 416.1131} C_DIS
LIN {X 78.8825,Y 57.0283,Z 99,A 31.4362,B 24.9175,C -2.098,E1 25.1287,E2 413.7775} C_DIS
LIN {X 76.9207,Y 59.6459,Z 99,A 33.1844,B 24.9176,C -2.0959,E1 25.1258,E2 412.0426} C_DIS
LIN {X 74.4029,Y 62.7597,Z 99,A 35.5396,B 24.9172,C -2.1014,E1 25.1216,E2 409.6854} C_DIS
LIN {X 69.4416,Y 68.2076,Z 99,A 39.9672,B 24.9162,C -2.1144,E1 25.1132,E2 405.2464} C_DIS
LIN {X 66.6401,Y 70.9467,Z 99,A 43.318,B 24.9125,C -2.1593,E1 25.1062,E2 401.8031} C_DIS
LIN {X 62.4578,Y 74.6556,Z 99,A 45.5469,B 24.9153,C -2.1249,E1 25.1016,E2 399.6642} C_DIS
LIN {X 56.2655,Y 79.427,Z 99,A 50.2128,B 24.9145,C -2.1355,E1 25.0912,E2 394.9903} C_DIS
LIN {X 52.8627,Y 81.7312,Z 99,A 52.5468,B 24.9145,C -2.1362,E1 25.0858,E2 392.6624} C_DIS
LIN {X 49.3264,Y 83.9125,Z 99,A 54.8333,B 24.9146,C -2.1339,E1 25.0804,E2 390.3885} C_DIS
LIN {X 46.0448,Y 85.7577,Z 99,A 57.0651,B 24.9143,C -2.1375,E1 25.0749,E2 388.1547} C_DIS
LIN {X 43.2846,Y 87.1825,Z 99,A 58.9395,B 24.914,C -2.1416,E1 25.0702,E2 386.2758} C_DIS
LIN {X 40.3665,Y 88.5723,Z 99,A 60.9739,B 24.9134,C -2.1487,E1 25.065,E2 384.2296} C_DIS
LIN {X 37.2005,Y 89.9485,Z 99,A 63.4224,B 24.912,C -2.1663,E1 25.0587,E2 381.7452} C_DIS
LIN {X 33.9604,Y 91.2213,Z 99,A 64.9386,B 24.9134,C -2.1485,E1 25.0548,E2 380.2744} C_DIS
LIN {X 28.1448,Y 93.1796,Z 99,A 68.6365,B 24.9129,C -2.1545,E1 25.045,E2 376.5692} C_DIS
LIN {X 24.6997,Y 94.1515,Z 99,A 70.7407,B 24.9129,C -2.1558,E1 25.0393,E2 374.4654} C_DIS
LIN {X 20.0128,Y 95.2577,Z 99,A 73.4559,B 24.9131,C -2.1529,E1 25.0319,E2 371.7606} C_DIS
LIN {X 16.9355,Y 95.8521,Z 99,A 75.2766,B 24.9131,C -2.1528,E1 25.0269,E2 369.9423} C_DIS
LIN {X 13.2475,Y 96.4316,Z 99,A 77.5934,B 24.9127,C -2.1577,E1 25.0205,E2 367.616} C_DIS
LIN {X 9.6784,Y 96.8549,Z 99,A 79.7008,B 24.9127,C -2.1577,E1 25.0147,E2 365.51} C_DIS
LIN {X 5.9449,Y 97.1559,Z 99,A 82.0043,B 24.9124,C -2.1613,E1 25.0082,E2 363.199} C_DIS
LIN {X 1.3348,Y 97.3281,Z 99,A 84.4753,B 24.9131,C -2.1523,E1 25.0014,E2 360.7499} C_DIS
LIN {X -3.1067,Y 97.2867,Z 99,A 87.2499,B 24.9127,C -2.1573,E1 24.9936,E2 357.9632} C_DIS
LIN {X -6.8688,Y 97.094,Z 99,A 89.5046,B 24.9127,C -2.1578,E1 24.9873,E2 355.7067} C_DIS
LIN {X -11.7125,Y 96.6298,Z 99,A 92.5406,B 24.9123,C -2.1623,E1 24.9789,E2 352.6582} C_DIS
LIN {X -15.8738,Y 96.0333,Z 99,A 94.7505,B 24.9132,C -2.1513,E1 24.9728,E2 350.4724} C_DIS
LIN {X -19.0962,Y 95.4459,Z 99,A 96.5221,B 24.9138,C -2.1443,E1 24.968,E2 348.7156} C_DIS
LIN {X -22.2737,Y 94.7542,Z 99,A 98.6955,B 24.9132,C -2.1516,E1 24.962,E2 346.5219} C_DIS
LIN {X -25.7574,Y 93.8672,Z 99,A 100.6341,B 24.9138,C -2.1433,E1 24.9568,E2 344.6003} C_DIS
LIN {X -28.2339,Y 93.153,Z 99,A 102.4323,B 24.9132,C -2.1514,E1 24.952,E2 342.7799} C_DIS
LIN {X -35.3107,Y 90.706,Z 99,A 106.4234,B 24.9148,C -2.1314,E1 24.9416,E2 338.8284} C_DIS
LIN {X -39.3501,Y 89.0268,Z 99,A 109.52,B 24.9137,C -2.1456,E1 24.9335,E2 335.6908} C_DIS
LIN {X -44.3619,Y 86.6393,Z 99,A 112.5193,B 24.9148,C -2.1312,E1 24.9261,E2 332.718} C_DIS
LIN {X -46.9616,Y 85.26,Z 99,A 114.8725,B 24.9133,C -2.1494,E1 24.9202,E2 330.3147} C_DIS
LIN {X -50.214,Y 83.385,Z 99,A 116.5716,B 24.9151,C -2.128,E1 24.9162,E2 328.6614} C_DIS
LIN {X -53.3581,Y 81.4084,Z 99,A 118.7084,B 24.9155,C -2.1222,E1 24.9112,E2 326.5316} C_DIS
LIN {X -56.3823,Y 79.3436,Z 99,A 121.0291,B 24.9155,C -2.1234,E1 24.9059,E2 324.2} C_DIS
LIN {X -61.0625,Y 75.8011,Z 99,A 124.3326,B 24.9164,C -2.111,E1 24.8986,E2 320.9141} C_DIS
LIN {X -63.4203,Y 73.8401,Z 99,A 126.4406,B 24.9159,C -2.1171,E1 24.8941,E2 318.7833} C_DIS
LIN {X -66.2417,Y 71.3206,Z 99,A 129.252,B 24.9148,C -2.1316,E1 24.8883,E2 315.9259} C_DIS
LIN {X -69.6923,Y 67.9532,Z 99,A 131.2298,B 24.9176,C -2.0958,E1 24.8845,E2 314.0249} C_DIS
LIN {X -73.2867,Y 64.0578,Z 99,A 134.3025,B 24.9184,C -2.0864,E1 24.8788,E2 310.961} C_DIS
LIN {X -76.7809,Y 59.8273,Z 99,A 137.6804,B 24.9186,C -2.0828,E1 24.8728,E2 307.5761} C_DIS
LIN {X -78.9997,Y 56.8643,Z 99,A 140.4633,B 24.9175,C -2.097,E1 24.8682,E2 304.7459} C_DIS
LIN {X -81.2447,Y 53.6063,Z 99,A 142.3846,B 24.9191,C -2.0769,E1 24.8652,E2 302.8627} C_DIS
LIN {X -83.3703,Y 50.2382,Z 99,A 144.5454,B 24.9201,C -2.0642,E1 24.8621,E2 300.7212} C_DIS
LIN {X -85.2508,Y 46.9781,Z 99,A 147.0071,B 24.92,C -2.0659,E1 24.8587,E2 298.2427} C_DIS
LIN {X -87.2515,Y 43.1453,Z 99,A 149.2643,B 24.9213,C -2.0489,E1 24.8559,E2 296.0138} C_DIS
LIN {X -89.0006,Y 39.4127,Z 99,A 151.9432,B 24.9213,C -2.0499,E1 24.8528,E2 293.3179} C_DIS
LIN {X -90.5214,Y 35.7808,Z 99,A 154.0934,B 24.9222,C -2.0373,E1 24.8505,E2 291.1858} C_DIS
LIN {X -91.7066,Y 32.6254,Z 99,A 155.9186,B 24.923,C -2.026,E1 24.8488,E2 289.3773} C_DIS
LIN {X -93.2512,Y 27.9036,Z 99,A 158.71,B 24.9241,C -2.0125,E1 24.8464,E2 286.6019} C_DIS
LIN {X -93.8982,Y 25.6415,Z 99,A 161.0352,B 24.922,C -2.0389,E1 24.8447,E2 284.2003} C_DIS
LIN {X -94.8413,Y 21.8967,Z 99,A 162.5568,B 24.9245,C -2.0071,E1 24.8437,E2 282.7458} C_DIS
LIN {X -95.45,Y 19.0677,Z 99,A 164.9455,B 24.9232,C -2.0241,E1 24.8424,E2 280.3024} C_DIS
LIN {X -96.0954,Y 15.5027,Z 99,A 166.8547,B 24.9243,C -2.0099,E1 24.8415,E2 278.4158} C_DIS
LIN {X -96.6588,Y 11.4647,Z 99,A 168.806,B 24.9259,C -1.9875,E1 24.8408,E2 276.5061} C_DIS
LIN {X -97.0614,Y 7.3216,Z 99,A 171.3852,B 24.9262,C -1.9838,E1 24.8402,E2 273.9203} C_DIS
LIN {X -97.2422,Y 4.2775,Z 99,A 173.254,B 24.9265,C -1.9804,E1 24.8399,E2 272.0483} C_DIS
LIN {X -97.332,Y 0.9994,Z 99,A 175.339,B 24.9265,C -1.9793,E1 24.8398,E2 269.9536} C_DIS
LIN {X -97.2944,Y -2.8562,Z 99,A 177.4686,B 24.9274,C -1.9674,E1 24.8398,E2 267.8394} C_DIS
LIN {X -97.1504,Y -6.0349,Z 99,A 179.441,B 24.9276,C -1.9647,E1 24.8402,E2 265.8617} C_DIS
LIN {X -96.8677,Y -9.5564,Z 99,A -178.4231,B 24.928,C -1.9599,E1 24.8407,E2 263.7244} C_DIS
LIN {X -96.4475,Y -13.1352,Z 99,A -176.2937,B 24.9285,C -1.9535,E1 24.8415,E2 261.5976} C_DIS
LIN {X -95.9541,Y -16.3476,Z 99,A -174.3872,B 24.9289,C -1.9473,E1 24.8423,E2 259.6946} C_DIS
LIN {X -95.3362,Y -19.6302,Z 99,A -172.4756,B 24.9295,C -1.9393,E1 24.8434,E2 257.7905} C_DIS
LIN {X -94.5526,Y -23.1114,Z 99,A -170.5793,B 24.9304,C -1.9262,E1 24.8446,E2 255.9145} C_DIS
LIN {X -93.3431,Y -27.5937,Z 99,A -167.7858,B 24.9309,C -1.9198,E1 24.8467,E2 253.12} C_DIS
LIN {X -91.7887,Y -32.3915,Z 99,A -164.532,B 24.9309,C -1.9203,E1 24.8495,E2 249.8464} C_DIS
LIN {X -90.542,Y -35.7282,Z 99,A -162.8073,B 24.9322,C -1.9019,E1 24.8512,E2 248.1558} C_DIS
LIN {X -89.3841,Y -38.5355,Z 99,A -160.6538,B 24.9317,C -1.9089,E1 24.8536,E2 245.9739} C_DIS
LIN {X -87.8735,Y -41.8652,Z 99,A -158.5717,B 24.9323,C -1.9005,E1 24.856,E2 243.9005} C_DIS
LIN {X -86.7688,Y -44.1085,Z 99,A -156.8453,B 24.932,C -1.9049,E1 24.8582,E2 242.1543} C_DIS
LIN {X -84.8471,Y -47.701,Z 99,A -154.8385,B 24.9334,C -1.8853,E1 24.8608,E2 240.1835} C_DIS
LIN {X -81.8618,Y -52.6593,Z 99,A -151.2142,B 24.9334,C -1.8835,E1 24.8662,E2 236.5448} C_DIS
LIN {X -79.9125,Y -55.5728,Z 99,A -149.2223,B 24.934,C -1.8759,E1 24.8693,E2 234.5613} C_DIS
LIN {X -76.7685,Y -59.8434,Z 99,A -145.9359,B 24.9342,C -1.8738,E1 24.8748,E2 231.2641} C_DIS
LIN {X -74.5952,Y -62.5306,Z 99,A -144.0591,B 24.9349,C -1.8637,E1 24.8781,E2 229.4027} C_DIS
LIN {X -72.4335,Y -65.0211,Z 99,A -141.6874,B 24.9342,C -1.874,E1 24.8826,E2 226.9959} C_DIS
LIN {X -69.9296,Y -67.707,Z 99,A -139.3229,B 24.934,C -1.8762,E1 24.8872,E2 224.6157} C_DIS
LIN {X -67.4216,Y -70.2046,Z 99,A -137.2189,B 24.9343,C -1.8726,E1 24.8914,E2 222.5116} C_DIS
LIN {X -64.778,Y -72.6511,Z 99,A -135.5572,B 24.9357,C -1.8527,E1 24.8948,E2 220.8909} C_DIS
LIN {X -62.824,Y -74.3481,Z 99,A -133.2563,B 24.934,C -1.8766,E1 24.8999,E2 218.5241} C_DIS
LIN {X -59.1657,Y -77.2907,Z 99,A -131.3255,B 24.9363,C -1.8428,E1 24.9039,E2 216.6668} C_DIS
LIN {X -55.8537,Y -79.7172,Z 99,A -128.8733,B 24.9365,C -1.8399,E1 24.9095,E2 214.2129} C_DIS
LIN {X -53.1787,Y -81.5267,Z 99,A -126.9202,B 24.9366,C -1.8387,E1 24.914,E2 212.2563} C_DIS
LIN {X -50.5108,Y -83.2046,Z 99,A -125.0591,B 24.9368,C -1.8361,E1 24.9185,E2 210.3954} C_DIS
LIN {X -47.4014,Y -85.0144,Z 99,A -122.9644,B 24.9371,C -1.8324,E1 24.9235,E2 208.3035} C_DIS
LIN {X -44.2385,Y -86.7024,Z 99,A -120.9248,B 24.9374,C -1.8272,E1 24.9286,E2 206.2706} C_DIS
LIN {X -41.1382,Y -88.2156,Z 99,A -118.1197,B 24.9357,C -1.8522,E1 24.9358,E2 203.3991} C_DIS
LIN {X -37.1467,Y -89.9706,Z 99,A -116.2439,B 24.9376,C -1.825,E1 24.9405,E2 201.5837} C_DIS
LIN {X -31.3882,Y -92.1369,Z 99,A -112.7311,B 24.9381,C -1.8178,E1 24.9497,E2 198.0806} C_DIS
LIN {X -28.7721,Y -92.9866,Z 99,A -111.065,B 24.9381,C -1.8183,E1 24.9541,E2 196.4105} C_DIS
LIN {X -26.2086,Y -93.742,Z 99,A -109.1302,B 24.9372,C -1.8302,E1 24.9594,E2 194.4443} C_DIS
LIN {X -21.9867,Y -94.8205,Z 99,A -106.9133,B 24.9382,C -1.8163,E1 24.9654,E2 192.2573} C_DIS
LIN {X -18.7907,Y -95.5061,Z 99,A -104.8427,B 24.9379,C -1.8208,E1 24.9711,E2 190.1737} C_DIS
LIN {X -15.8635,Y -96.035,Z 99,A -103.1812,B 24.9381,C -1.817,E1 24.9756,E2 188.5196} C_DIS
LIN {X -11.9396,Y -96.6029,Z 99,A -100.7628,B 24.9379,C -1.8196,E1 24.9823,E2 186.0933} C_DIS
LIN {X -8.2723,Y -96.9855,Z 99,A -98.8561,B 24.9386,C -1.8098,E1 24.9876,E2 184.2086} C_DIS
LIN {X -4.5831,Y -97.2291,Z 99,A -96.544,B 24.9383,C -1.8149,E1 24.9941,E2 181.8838} C_DIS
LIN {X 0.6795,Y -97.3292,Z 99,A -94.8341,B 24.9416,C -1.7652,E1 24.9986,E2 180.2914} C_DIS
Enddeposition()
LIN {X 0.6795,Y -97.3292,Z 99,A -94.8341,B 24.9416,C -1.7652,E1 24.9986,E2 180.2914} C_DIS
Startdeposition()
$VEL.CP = VEL_PRINT
LIN {X -0.103,Y -96.4509,Z 99,A -94.9881,B 24.9398,C -1.7918,E1 24.9983,E2 180.3825} C_DIS
LIN {X -4.3836,Y -96.3504,Z 99,A -97.3548,B 24.9394,C -1.7978,E1 24.9917,E2 182.7354} C_DIS
LIN {X -7.9102,Y -96.1251,Z 99,A -99.4987,B 24.9395,C -1.7962,E1 24.9857,E2 184.8838} C_DIS
LIN {X -11.3695,Y -95.7774,Z 99,A -101.3224,B 24.9389,C -1.805,E1 24.9807,E2 186.6878} C_DIS
LIN {X -14.2582,Y -95.3912,Z 99,A -103.2068,B 24.9393,C -1.8,E1 24.9754,E2 188.5857} C_DIS
LIN {X -17.2847,Y -94.8885,Z 99,A -105.1516,B 24.9395,C -1.7963,E1 24.9701,E2 190.5411} C_DIS
LIN {X -21.085,Y -94.1184,Z 99,A -107.4997,B 24.9395,C -1.7957,E1 24.9636,E2 192.8933} C_DIS
LIN {X -23.9144,Y -93.438,Z 99,A -109.0903,B 24.9392,C -1.8015,E1 24.9594,E2 194.4725} C_DIS
LIN {X -27.3855,Y -92.4802,Z 99,A -111.246,B 24.9392,C -1.8024,E1 24.9536,E2 196.6297} C_DIS
LIN {X -30.3967,Y -91.5357,Z 99,A -112.9205,B 24.9385,C -1.8107,E1 24.9491,E2 198.2874} C_DIS
LIN {X -33.4577,Y -90.4617,Z 99,A -115.1344,B 24.9391,C -1.8025,E1 24.9433,E2 200.5251} C_DIS
LIN {X -36.6935,Y -89.1979,Z 99,A -117.0133,B 24.9385,C -1.8109,E1 24.9384,E2 202.3882} C_DIS
LIN {X -40.1538,Y -87.6958,Z 99,A -119.2619,B 24.9384,C -1.813,E1 24.9327,E2 204.6372} C_DIS
LIN {X -42.8433,Y -86.4118,Z 99,A -121.1178,B 24.9384,C -1.8123,E1 24.928,E2 206.4996} C_DIS
LIN {X -45.727,Y -84.9216,Z 99,A -123.1369,B 24.9384,C -1.8117,E1 24.923,E2 208.5258} C_DIS
LIN {X -48.9313,Y -83.1162,Z 99,A -125.2611,B 24.9381,C -1.8168,E1 24.9179,E2 210.644} C_DIS
LIN {X -51.8214,Y -81.3462,Z 99,A -127.2892,B 24.938,C -1.8193,E1 24.9131,E2 212.6725} C_DIS
LIN {X -54.6043,Y -79.5061,Z 99,A -129.3679,B 24.938,C -1.8193,E1 24.9082,E2 214.7584} C_DIS
LIN {X -57.6284,Y -77.3412,Z 99,A -131.3772,B 24.9372,C -1.8297,E1 24.9037,E2 216.7497} C_DIS
LIN {X -60.7153,Y -74.9413,Z 99,A -133.8223,B 24.9372,C -1.8299,E1 24.8984,E2 219.2035} C_DIS
LIN {X -63.3204,Y -72.7537,Z 99,A -135.8386,B 24.937,C -1.8339,E1 24.8941,E2 221.2181} C_DIS
LIN {X -66.9686,Y -69.4101,Z 99,A -139.3062,B 24.9377,C -1.8225,E1 24.8869,E2 224.7271} C_DIS
LIN {X -69.3888,Y -66.9907,Z 99,A -140.4503,B 24.9354,C -1.8561,E1 24.8849,E2 225.7959} C_DIS
LIN {X -71.7661,Y -64.4375,Z 99,A -142.9004,B 24.936,C -1.8482,E1 24.8802,E2 228.2757} C_DIS
LIN {X -73.8962,Y -61.9846,Z 99,A -144.9691,B 24.936,C -1.8481,E1 24.8764,E2 230.3541} C_DIS
LIN {X -76.1959,Y -59.1342,Z 99,A -147.0813,B 24.9355,C -1.8553,E1 24.8727,E2 232.459} C_DIS
LIN {X -78.2745,Y -56.3545,Z 99,A -149.0396,B 24.9349,C -1.8638,E1 24.8695,E2 234.4066} C_DIS
LIN {X -79.8927,Y -54.0344,Z 99,A -150.7898,B 24.9347,C -1.8658,E1 24.8667,E2 236.1607} C_DIS
LIN {X -83.5198,Y -48.2393,Z 99,A -154.905,B 24.9341,C -1.8746,E1 24.8607,E2 240.2758} C_DIS
LIN {X -85.8435,Y -43.971,Z 99,A -157.8367,B 24.9337,C -1.8811,E1 24.8569,E2 243.2077} C_DIS
LIN {X -87.4439,Y -40.6954,Z 99,A -159.9988,B 24.9332,C -1.8873,E1 24.8543,E2 245.3668} C_DIS
LIN {X -88.6499,Y -38.0011,Z 99,A -161.6973,B 24.9328,C -1.894,E1 24.8524,E2 247.0585} C_DIS
LIN {X -89.7675,Y -35.2752,Z 99,A -163.3934,B 24.9323,C -1.9009,E1 24.8506,E2 248.7478} C_DIS
LIN {X -90.7634,Y -32.6305,Z 99,A -165.0881,B 24.9319,C -1.9053,E1 24.849,E2 250.4415} C_DIS
LIN {X -91.9195,Y -29.2165,Z 99,A -167.4611,B 24.932,C -1.9042,E1 24.8469,E2 252.8306} C_DIS
LIN {X -92.8632,Y -26.0583,Z 99,A -169.2031,B 24.9311,C -1.9171,E1 24.8455,E2 254.552} C_DIS
LIN {X -93.7397,Y -22.7033,Z 99,A -171.4586,B 24.9311,C -1.9171,E1 24.844,E2 256.8205} C_DIS
LIN {X -94.5953,Y -18.8312,Z 99,A -173.7853,B 24.9305,C -1.9253,E1 24.8426,E2 259.1414} C_DIS
LIN {X -95.1524,Y -15.7669,Z 99,A -175.7077,B 24.9302,C -1.9289,E1 24.8417,E2 261.0668} C_DIS
LIN {X -95.6647,Y -12.2812,Z 99,A -177.6957,B 24.9295,C -1.9388,E1 24.841,E2 263.0429} C_DIS
LIN {X -96.0289,Y -9.0006,Z 99,A -179.7194,B 24.9292,C -1.943,E1 24.8404,E2 265.0688} C_DIS
LIN {X -96.2642,Y -6.0014,Z 99,A 178.3357,B 24.9292,C -1.9437,E1 24.84,E2 267.0237} C_DIS
LIN {X -96.427,Y -2.1203,Z 99,A 176.123,B 24.9284,C -1.9541,E1 24.8398,E2 269.2249} C_DIS
LIN {X -96.4385,Y 1.4962,Z 99,A 173.9482,B 24.928,C -1.9602,E1 24.8398,E2 271.3983} C_DIS
LIN {X -96.3457,Y 4.4931,Z 99,A 172.3081,B 24.9272,C -1.9704,E1 24.84,E2 273.0239} C_DIS
LIN {X -96.1619,Y 7.4491,Z 99,A 170.5296,B 24.9268,C -1.9754,E1 24.8403,E2 274.801} C_DIS
LIN {X -95.8429,Y 10.81,Z 99,A 168.3547,B 24.9268,C -1.9765,E1 24.841,E2 276.9864} C_DIS
LIN {X -95.0104,Y 16.607,Z 99,A 164.4435,B 24.9269,C -1.9741,E1 24.8427,E2 280.9267} C_DIS
LIN {X -94.4002,Y 19.7816,Z 99,A 162.9121,B 24.9256,C -1.9924,E1 24.8435,E2 282.4234} C_DIS
LIN {X -93.8831,Y 22.1061,Z 99,A 161.0419,B 24.9263,C -1.9826,E1 24.8447,E2 284.3281} C_DIS
LIN {X -93.0511,Y 25.3789,Z 99,A 159.4547,B 24.9248,C -2.0021,E1 24.8459,E2 285.8779} C_DIS
LIN {X -92.1982,Y 28.3214,Z 99,A 157.5879,B 24.9245,C -2.0063,E1 24.8474,E2 287.7454} C_DIS
LIN {X -90.9465,Y 32.1142,Z 99,A 155.3648,B 24.9236,C -2.0184,E1 24.8493,E2 289.9523} C_DIS
LIN {X -89.8066,Y 35.1757,Z 99,A 153.3453,B 24.9233,C -2.0219,E1 24.8513,E2 291.9748} C_DIS
LIN {X -88.4507,Y 38.4582,Z 99,A 151.2048,B 24.9229,C -2.0273,E1 24.8537,E2 294.1143} C_DIS
LIN {X -87.0721,Y 41.4862,Z 99,A 149.2002,B 24.9225,C -2.0324,E1 24.856,E2 296.1178} C_DIS
LIN {X -85.555,Y 44.5322,Z 99,A 147.2486,B 24.9219,C -2.0405,E1 24.8585,E2 298.0603} C_DIS
LIN {X -84.1222,Y 47.181,Z 99,A 145.3124,B 24.9219,C -2.0411,E1 24.8611,E2 300.0055} C_DIS
LIN {X -82.5513,Y 49.8789,Z 99,A 143.4828,B 24.9214,C -2.0472,E1 24.8637,E2 301.8299} C_DIS
LIN {X -80.9164,Y 52.491,Z 99,A 141.5275,B 24.9214,C -2.0483,E1 24.8667,E2 303.7924} C_DIS
LIN {X -78.6658,Y 55.8059,Z 99,A 139.4165,B 24.9201,C -2.0635,E1 24.87,E2 305.8776} C_DIS
LIN {X -77.0167,Y 58.0603,Z 99,A 137.5294,B 24.9204,C -2.0607,E1 24.8731,E2 307.7805} C_DIS
LIN {X -74.3897,Y 61.3907,Z 99,A 134.642,B 24.9208,C -2.0555,E1 24.8783,E2 310.6937} C_DIS
LIN {X -72.2475,Y 63.8998,Z 99,A 132.9894,B 24.9196,C -2.0703,E1 24.8813,E2 312.3184} C_DIS
LIN {X -69.7338,Y 66.6328,Z 99,A 130.8466,B 24.919,C -2.0779,E1 24.8853,E2 314.4527} C_DIS
LIN {X -66.6889,Y 69.6795,Z 99,A 128.0967,B 24.919,C -2.0779,E1 24.8908,E2 317.2142} C_DIS
LIN {X -63.6065,Y 72.5038,Z 99,A 125.7896,B 24.9181,C -2.0892,E1 24.8956,E2 319.5033} C_DIS
LIN {X -60.8223,Y 74.8546,Z 99,A 123.7053,B 24.9176,C -2.0966,E1 24.9001,E2 321.5779} C_DIS
LIN {X -58.3251,Y 76.8178,Z 99,A 121.7091,B 24.9176,C -2.097,E1 24.9045,E2 323.5804} C_DIS
LIN {X -55.5572,Y 78.8425,Z 99,A 119.8604,B 24.9167,C -2.1074,E1 24.9086,E2 325.411} C_DIS
LIN {X -53.1094,Y 80.5105,Z 99,A 117.9698,B 24.9167,C -2.1065,E1 24.913,E2 327.3099} C_DIS
LIN {X -50.1738,Y 82.372,Z 99,A 115.882,B 24.9165,C -2.1096,E1 24.918,E2 329.3969} C_DIS
LIN {X -46.8247,Y 84.3211,Z 99,A 113.5023,B 24.9165,C -2.1111,E1 24.9238,E2 331.7801} C_DIS
LIN {X -44.0981,Y 85.7786,Z 99,A 110.9256,B 24.9181,C -2.0898,E1 24.9303,E2 334.4144} C_DIS
LIN {X -40.0348,Y 87.7495,Z 99,A 109.0633,B 24.9156,C -2.121,E1 24.9348,E2 336.2073} C_DIS
LIN {X -37.1718,Y 88.9995,Z 99,A 107.1525,B 24.9156,C -2.1218,E1 24.9397,E2 338.1205} C_DIS
LIN {X -35.0399,Y 89.8599,Z 99,A 105.2218,B 24.9169,C -2.1048,E1 24.9449,E2 340.0958} C_DIS
LIN {X -31.5908,Y 91.1295,Z 99,A 103.3754,B 24.9158,C -2.1188,E1 24.9497,E2 341.9126} C_DIS
LIN {X -26.7005,Y 92.6812,Z 99,A 100.6972,B 24.9145,C -2.1347,E1 24.9567,E2 344.5576} C_DIS
LIN {X -24.0158,Y 93.4119,Z 99,A 98.9271,B 24.9147,C -2.1324,E1 24.9615,E2 346.3359} C_DIS
LIN {X -20.7632,Y 94.1886,Z 99,A 97.0557,B 24.9143,C -2.1381,E1 24.9666,E2 348.196} C_DIS
LIN {X -18.0252,Y 94.7507,Z 99,A 95.143,B 24.9148,C -2.1309,E1 24.9719,E2 350.1281} C_DIS
LIN {X -14.1653,Y 95.4056,Z 99,A 92.8135,B 24.9148,C -2.1323,E1 24.9783,E2 352.4563} C_DIS
LIN {X -10.3954,Y 95.8885,Z 99,A 90.6674,B 24.9143,C -2.1375,E1 24.9842,E2 354.5916} C_DIS
LIN {X -7.2373,Y 96.1789,Z 99,A 88.6379,B 24.9146,C -2.1333,E1 24.9899,E2 356.6319} C_DIS
LIN {X -3.5165,Y 96.3872,Z 99,A 86.5861,B 24.9141,C -2.1397,E1 24.9956,E2 358.669} C_DIS
LIN {X -0.2819,Y 96.4498,Z 99,A 84.6391,B 24.9141,C -2.1393,E1 25.001,E2 360.6171} C_DIS
LIN {X 2.7045,Y 96.4121,Z 99,A 82.7919,B 24.9144,C -2.137,E1 25.0062,E2 362.4694} C_DIS
LIN {X 6.5013,Y 96.2304,Z 99,A 80.6084,B 24.9141,C -2.1396,E1 25.0123,E2 364.6459} C_DIS
LIN {X 9.4223,Y 95.99,Z 99,A 78.7951,B 24.9144,C -2.1369,E1 25.0173,E2 366.4645} C_DIS
LIN {X 12.8649,Y 95.5891,Z 99,A 76.7018,B 24.9144,C -2.1353,E1 25.0231,E2 368.5601} C_DIS
LIN {X 16.5035,Y 95.029,Z 99,A 74.6059,B 24.9143,C -2.1377,E1 25.0289,E2 370.648} C_DIS
LIN {X 19.6337,Y 94.4305,Z 99,A 72.9413,B 24.9137,C -2.145,E1 25.0334,E2 372.2933} C_DIS
LIN {X 22.2602,Y 93.8475,Z 99,A 70.9657,B 24.9148,C -2.1308,E1 25.0389,E2 374.3} C_DIS
LIN {X 26.1147,Y 92.8472,Z 99,A 68.7353,B 24.9146,C -2.1341,E1 25.0448,E2 376.519} C_DIS
LIN {X 30.2656,Y 91.5798,Z 99,A 66.2271,B 24.9146,C -2.1346,E1 25.0515,E2 379.0215} C_DIS
LIN {X 33.0218,Y 90.6207,Z 99,A 64.5021,B 24.9146,C -2.1334,E1 25.056,E2 380.7459} C_DIS
LIN {X 36.3457,Y 89.3394,Z 99,A 62.3664,B 24.9149,C -2.1305,E1 25.0616,E2 382.8835} C_DIS
LIN {X 39.6354,Y 87.9294,Z 99,A 60.2963,B 24.9149,C -2.1302,E1 25.0669,E2 384.9493} C_DIS
LIN {X 42.3224,Y 86.67,Z 99,A 58.3711,B 24.9155,C -2.1222,E1 25.0718,E2 386.8885} C_DIS
LIN {X 45.1725,Y 85.2177,Z 99,A 56.6435,B 24.9152,C -2.126,E1 25.076,E2 388.6023} C_DIS
LIN {X 48.0683,Y 83.6181,Z 99,A 54.7893,B 24.9152,C -2.1273,E1 25.0805,E2 390.4479} C_DIS
LIN {X 50.5949,Y 82.1161,Z 99,A 52.8095,B 24.916,C -2.1161,E1 25.0853,E2 392.448} C_DIS
LIN {X 53.008,Y 80.5773,Z 99,A 51.1555,B 24.916,C -2.1151,E1 25.0892,E2 394.0989} C_DIS
LIN {X 55.7166,Y 78.7296,Z 99,A 48.3168,B 24.9189,C -2.0793,E1 25.0958,E2 397.0124} C_DIS
LIN {X 59.667,Y 75.7788,Z 99,A 46.2939,B 24.9167,C -2.1072,E1 25.1001,E2 398.962} C_DIS
LIN {X 62.4287,Y 73.5203,Z 99,A 44.2402,B 24.9169,C -2.1056,E1 25.1045,E2 401.0116} C_DIS
LIN {X 66.2667,Y 70.081,Z 99,A 41.0573,B 24.9177,C -2.0949,E1 25.1111,E2 404.207} C_DIS
LIN {X 68.4621,Y 67.9378,Z 99,A 38.5661,B 24.9199,C -2.0663,E1 25.1161,E2 406.7553} C_DIS
LIN {X 71.5447,Y 64.6848,Z 99,A 36.6463,B 24.9183,C -2.0878,E1 25.1196,E2 408.6157} C_DIS
LIN {X 73.6836,Y 62.237,Z 99,A 34.5133,B 24.9192,C -2.0758,E1 25.1235,E2 410.7673} C_DIS
LIN {X 76.2577,Y 59.054,Z 99,A 32.3168,B 24.919,C -2.0788,E1 25.1273,E2 412.9464} C_DIS
LIN {X 78.3133,Y 56.3,Z 99,A 30.2404,B 24.9195,C -2.0724,E1 25.1307,E2 415.0279} C_DIS
LIN {X 80.3177,Y 53.4018,Z 99,A 28.1337,B 24.9199,C -2.0666,E1 25.134,E2 417.138} C_DIS
LIN {X 82.5944,Y 49.8078,Z 99,A 25.675,B 24.9202,C -2.0626,E1 25.1377,E2 419.5938} C_DIS
LIN {X 84.3835,Y 46.7129,Z 99,A 23.5695,B 24.9206,C -2.0575,E1 25.1406,E2 421.7002} C_DIS
LIN {X 85.7759,Y 44.1034,Z 99,A 21.8369,B 24.9209,C -2.0536,E1 25.1428,E2 423.4329} C_DIS
LIN {X 87.3,Y 41.0044,Z 99,A 19.4843,B 24.9222,C -2.0364,E1 25.1457,E2 425.8134} C_DIS
LIN {X 89.1946,Y 36.7016,Z 99,A 17.1075,B 24.9216,C -2.0442,E1 25.1482,E2 428.1588} C_DIS
LIN {X 90.1837,Y 34.1973,Z 99,A 15.4758,B 24.9221,C -2.0383,E1 25.1499,E2 429.7953} C_DIS
LIN {X 91.682,Y 29.9504,Z 99,A 12.9562,B 24.9222,C -2.0363,E1 25.1522,E2 432.3055} C_DIS
LIN {X 92.5988,Y 26.9855,Z 99,A 10.8937,B 24.9233,C -2.0223,E1 25.1538,E2 434.3893} C_DIS
LIN {X 93.4225,Y 23.9748,Z 99,A 9.1859,B 24.9233,C -2.0223,E1 25.1551,E2 436.0874} C_DIS
LIN {X 94.2143,Y 20.645,Z 99,A 7.1103,B 24.9239,C -2.0144,E1 25.1564,E2 438.1696} C_DIS
LIN {X 94.7978,Y 17.7803,Z 99,A 5.3293,B 24.9245,C -2.0072,E1 25.1573,E2 439.957} C_DIS
LIN {X 95.2457,Y 15.1994,Z 99,A 4.0062,B 24.9241,C -2.0113,E1 25.1579,E2 441.2627} C_DIS
LIN {X 95.6915,Y 12.0744,Z 99,A 1.9747,B 24.925,C -1.9994,E1 25.1587,E2 443.3104} C_DIS
LIN {X 96.0031,Y 9.2802,Z 99,A 0.2786,B 24.9255,C -1.993,E1 25.1592,E2 445.0114} C_DIS
LIN {X 96.2168,Y 6.7013,Z 99,A -1.195,B 24.9257,C -1.9906,E1 25.1595,E2 446.482} C_DIS
LIN {X 96.3944,Y 3.2834,Z 99,A -2.9652,B 24.9254,C -1.9942,E1 25.1597,E2 448.233} C_DIS
LIN {X 96.4462,Y 0.879,Z 99,A -4.702,B 24.9267,C -1.9777,E1 25.1597,E2 449.9985} C_DIS
LIN {X 96.4096,Y -2.7876,Z 99,A -6.8318,B 24.927,C -1.9726,E1 25.1597,E2 452.1277} C_DIS
LIN {X 96.2597,Y -6.0669,Z 99,A -8.718,B 24.9273,C -1.9687,E1 25.1594,E2 454.0118} C_DIS
LIN {X 96.02,Y -9.0975,Z 99,A -10.6087,B 24.928,C -1.9596,E1 25.1589,E2 455.9127} C_DIS
LIN {X 95.6215,Y -12.6149,Z 99,A -12.5392,B 24.928,C -1.9596,E1 25.1583,E2 457.8321} C_DIS
LIN {X 95.1771,Y -15.6188,Z 99,A -14.3939,B 24.9286,C -1.9518,E1 25.1575,E2 459.6943} C_DIS
LIN {X 94.5758,Y -18.9263,Z 99,A -16.3973,B 24.9291,C -1.9451,E1 25.1564,E2 461.7016} C_DIS
LIN {X 93.8379,Y -22.3007,Z 99,A -18.459,B 24.9296,C -1.9382,E1 25.1552,E2 463.7677} C_DIS
LIN {X 93.032,Y -25.4499,Z 99,A -20.2446,B 24.9296,C -1.9377,E1 25.1539,E2 465.5442} C_DIS
LIN {X 92.4071,Y -27.6319,Z 99,A -22.5978,B 24.9327,C -1.8949,E1 25.1519,E2 467.9848} C_DIS
LIN {X 90.8682,Y -32.3374,Z 99,A -24.6846,B 24.931,C -1.9184,E1 25.1501,E2 470.0045} C_DIS
LIN {X 89.5656,Y -35.7893,Z 99,A -26.6837,B 24.931,C -1.9191,E1 25.1481,E2 471.9909} C_DIS
LIN {X 88.3722,Y -38.6381,Z 99,A -28.694,B 24.9318,C -1.9067,E1 25.1458,E2 474.0193} C_DIS
LIN {X 87.0659,Y -41.4991,Z 99,A -30.4574,B 24.932,C -1.9051,E1 25.1438,E2 475.777} C_DIS
LIN {X 85.8724,Y -43.9144,Z 99,A -32.566,B 24.9337,C -1.8809,E1 25.141,E2 477.9315} C_DIS
LIN {X 84.2429,Y -46.9647,Z 99,A -34.0961,B 24.9327,C -1.8949,E1 25.139,E2 479.4206} C_DIS
LIN {X 82.6854,Y -49.6582,Z 99,A -36.036,B 24.9333,C -1.8861,E1 25.1363,E2 481.3714} C_DIS
LIN {X 80.6855,Y -52.8441,Z 99,A -38.1959,B 24.9336,C -1.8826,E1 25.133,E2 483.5286} C_DIS
LIN {X 79.0336,Y -55.284,Z 99,A -40.8576,B 24.9363,C -1.8432,E1 25.1286,E2 486.2704} C_DIS
LIN {X 75.9722,Y -59.4223,Z 99,A -42.968,B 24.9344,C -1.8708,E1 25.1252,E2 488.3055} C_DIS
LIN {X 73.7576,Y -62.1501,Z 99,A -45.117,B 24.9349,C -1.863,E1 25.1213,E2 490.4632} C_DIS
LIN {X 71.4391,Y -64.8021,Z 99,A -47.1509,B 24.9352,C -1.8599,E1 25.1175,E2 492.4953} C_DIS
LIN {X 69.3019,Y -67.0809,Z 99,A -49.0409,B 24.9356,C -1.854,E1 25.1139,E2 494.391} C_DIS
LIN {X 66.7632,Y -69.608,Z 99,A -51.1406,B 24.9359,C -1.8499,E1 25.1097,E2 496.4916} C_DIS
LIN {X 64.0269,Y -72.1337,Z 99,A -53.3371,B 24.9362,C -1.8453,E1 25.1051,E2 498.6901} C_DIS
LIN {X 61.6069,Y -74.2102,Z 99,A -55.2098,B 24.9364,C -1.8419,E1 25.1011,E2 500.5636} C_DIS
LIN {X 58.6427,Y -76.5746,Z 99,A -58.1407,B 24.9385,C -1.8117,E1 25.0945,E2 503.5552} C_DIS
LIN {X 55.1323,Y -79.1391,Z 99,A -59.9783,B 24.9369,C -1.8342,E1 25.0905,E2 505.3332} C_DIS
LIN {X 52.0506,Y -81.199,Z 99,A -62.1334,B 24.9371,C -1.8316,E1 25.0854,E2 507.4873} C_DIS
LIN {X 49.5916,Y -82.7258,Z 99,A -64.0227,B 24.9378,C -1.822,E1 25.0809,E2 509.3933} C_DIS
LIN {X 46.1359,Y -84.6998,Z 99,A -66.2228,B 24.9376,C -1.824,E1 25.0756,E2 511.5824} C_DIS
LIN {X 42.9786,Y -86.3447,Z 99,A -68.3683,B 24.938,C -1.8193,E1 25.0702,E2 513.733} C_DIS
LIN {X 40.1831,Y -87.6824,Z 99,A -70.2892,B 24.9384,C -1.8134,E1 25.0653,E2 515.6629} C_DIS
LIN {X 36.906,Y -89.1107,Z 99,A -72.2017,B 24.938,C -1.8181,E1 25.0605,E2 517.5598} C_DIS
LIN {X 34.9547,Y -89.8934,Z 99,A -73.7439,B 24.9389,C -1.8056,E1 25.0564,E2 519.1282} C_DIS
LIN {X 30.7839,Y -91.4051,Z 99,A -76.0266,B 24.9382,C -1.8152,E1 25.0504,E2 521.3836} C_DIS
LIN {X 28.1048,Y -92.2654,Z 99,A -77.9366,B 24.939,C -1.8044,E1 25.0453,E2 523.3156} C_DIS
LIN {X 24.6176,Y -93.2568,Z 99,A -79.9486,B 24.9388,C -1.8073,E1 25.0399,E2 525.3176} C_DIS
LIN {X 21.7934,Y -93.9553,Z 99,A -81.6824,B 24.9389,C -1.8054,E1 25.0352,E2 527.0532} C_DIS
LIN {X 18.7799,Y -94.6053,Z 99,A -83.598,B 24.9392,C -1.8007,E1 25.0299,E2 528.9777} C_DIS
LIN {X 15.3489,Y -95.2223,Z 99,A -85.6915,B 24.9394,C -1.7983,E1 25.0241,E2 531.0746} C_DIS
LIN {X 11.7432,Y -95.7336,Z 99,A -87.5972,B 24.9389,C -1.8062,E1 25.0189,E2 532.9601} C_DIS
LIN {X 9.4189,Y -95.9897,Z 99,A -89.4386,B 24.94,C -1.7892,E1 25.0137,E2 534.8407} C_DIS
LIN {X 4.9558,Y -96.323,Z 99,A -91.8824,B 24.9396,C -1.7957,E1 25.0069,E2 537.2679} C_DIS
LIN {X 1.0581,Y -96.445,Z 99,A -93.9799,B 24.9391,C -1.8028,E1 25.0011,E2 539.3481} C_DIS
LIN {X 1.0581,Y -96.445,Z 99,A -93.9799,B 24.9391,C -1.8028,E1 25.0011,E2 539.3481} C_DIS
Enddeposition()
LIN {X 0.6729,Y -95.56,Z 99,A -94.1705,B 24.9379,C -1.8197,E1 25.0007,E2 539.4987} C_DIS
Startdeposition()
$VEL.CP = VEL_PRINT
LIN {X 4.0187,Y -95.4787,Z 99,A -91.5065,B 24.9363,C -1.8438,E1 25.0083,E2 536.7781} C_DIS
LIN {X 7.006,Y -95.3077,Z 99,A -89.8086,B 24.9365,C -1.8411,E1 25.013,E2 535.0873} C_DIS
LIN {X 10.4898,Y -94.9873,Z 99,A -87.7152,B 24.9364,C -1.8421,E1 25.0188,E2 532.9928} C_DIS
LIN {X 12.5855,Y -94.7314,Z 99,A -86.4166,B 24.9363,C -1.8441,E1 25.0224,E2 531.6906} C_DIS
LIN {X 15.1717,Y -94.353,Z 99,A -84.8824,B 24.9363,C -1.8441,E1 25.0267,E2 530.158} C_DIS
LIN {X 17.7454,Y -93.9017,Z 99,A -83.1832,B 24.9358,C -1.8502,E1 25.0314,E2 528.4462} C_DIS
LIN {X 20.662,Y -93.3033,Z 99,A -81.5033,B 24.936,C -1.8479,E1 25.0359,E2 526.7737} C_DIS
LIN {X 22.954,Y -92.7661,Z 99,A -80.0983,B 24.936,C -1.8491,E1 25.0398,E2 525.3681} C_DIS
LIN {X 25.4841,Y -92.1045,Z 99,A -78.563,B 24.9359,C -1.8495,E1 25.0439,E2 523.8342} C_DIS
LIN {X 27.732,Y -91.4527,Z 99,A -77.1639,B 24.9358,C -1.8509,E1 25.0476,E2 522.4341} C_DIS
LIN {X 30.8117,Y -90.4602,Z 99,A -75.0249,B 24.9351,C -1.8607,E1 25.0534,E2 520.276} C_DIS
LIN {X 34.1501,Y -89.2536,Z 99,A -73.0724,B 24.9354,C -1.857,E1 25.0584,E2 518.3364} C_DIS
LIN {X 37.4062,Y -87.9387,Z 99,A -71.007,B 24.9352,C -1.8586,E1 25.0638,E2 516.272} C_DIS
LIN {X 39.5483,Y -86.9963,Z 99,A -69.5798,B 24.935,C -1.8616,E1 25.0674,E2 514.8412} C_DIS
LIN {X 41.9143,Y -85.8828,Z 99,A -68.0485,B 24.935,C -1.8628,E1 25.0713,E2 513.3113} C_DIS
LIN {X 45.0402,Y -84.2855,Z 99,A -65.9486,B 24.9347,C -1.8661,E1 25.0765,E2 511.2092} C_DIS
LIN {X 46.8506,Y -83.2913,Z 99,A -64.6851,B 24.9345,C -1.8693,E1 25.0796,E2 509.942} C_DIS
LIN {X 49.1358,Y -81.9655,Z 99,A -62.9175,B 24.9338,C -1.8791,E1 25.0839,E2 508.1566} C_DIS
LIN {X 52.1026,Y -80.1123,Z 99,A -61.0512,B 24.9341,C -1.8744,E1 25.0882,E2 506.3074} C_DIS
LIN {X 54.7728,Y -78.3093,Z 99,A -59.0943,B 24.9338,C -1.8793,E1 25.0927,E2 504.3457} C_DIS
LIN {X 57.0979,Y -76.6309,Z 99,A -57.2714,B 24.9333,C -1.8868,E1 25.0969,E2 502.5115} C_DIS
LIN {X 59.721,Y -74.606,Z 99,A -55.2238,B 24.9328,C -1.8934,E1 25.1014,E2 500.4559} C_DIS
LIN {X 62.422,Y -72.3614,Z 99,A -53.1271,B 24.9325,C -1.8978,E1 25.1058,E2 498.357} C_DIS
LIN {X 65.0387,Y -70.0188,Z 99,A -51.0322,B 24.9322,C -1.9023,E1 25.1102,E2 496.2598} C_DIS
LIN {X 67.5595,Y -67.5897,Z 99,A -48.9407,B 24.9318,C -1.9071,E1 25.1143,E2 494.1657} C_DIS
LIN {X 70.0172,Y -65.0405,Z 99,A -46.8325,B 24.9315,C -1.9118,E1 25.1184,E2 492.0556} C_DIS
LIN {X 72.3597,Y -62.4238,Z 99,A -44.7388,B 24.9311,C -1.9168,E1 25.1222,E2 489.9596} C_DIS
LIN {X 74.5182,Y -59.8294,Z 99,A -42.8583,B 24.9311,C -1.9166,E1 25.1255,E2 488.0882} C_DIS
LIN {X 76.7766,Y -56.9033,Z 99,A -40.7333,B 24.931,C -1.9191,E1 25.1291,E2 485.9674} C_DIS
LIN {X 77.9919,Y -55.2242,Z 99,A -39.4669,B 24.9306,C -1.9235,E1 25.1312,E2 484.6969} C_DIS
LIN {X 79.4688,Y -53.0789,Z 99,A -37.953,B 24.9305,C -1.926,E1 25.1335,E2 483.1845} C_DIS
LIN {X 81.2144,Y -50.3652,Z 99,A -36.0278,B 24.9301,C -1.9311,E1 25.1364,E2 481.2569} C_DIS
LIN {X 82.42,Y -48.367,Z 99,A -34.6375,B 24.9298,C -1.9348,E1 25.1384,E2 479.865} C_DIS
LIN {X 83.7094,Y -46.1018,Z 99,A -33.0881,B 24.9295,C -1.9388,E1 25.1405,E2 478.3142} C_DIS
LIN {X 85.3388,Y -43.0106,Z 99,A -31.0125,B 24.9291,C -1.9443,E1 25.1432,E2 476.2367} C_DIS
LIN {X 86.7675,Y -40.0477,Z 99,A -29.014,B 24.9286,C -1.9513,E1 25.1456,E2 474.2326} C_DIS
LIN {X 87.832,Y -37.659,Z 99,A -27.4853,B 24.9284,C -1.9545,E1 25.1473,E2 472.7046} C_DIS
LIN {X 88.7279,Y -35.4967,Z 99,A -26.0933,B 24.9281,C -1.9584,E1 25.1488,E2 471.3111} C_DIS
LIN {X 89.8753,Y -32.4782,Z 99,A -24.1741,B 24.9277,C -1.9637,E1 25.1507,E2 469.3899} C_DIS
LIN {X 90.6999,Y -30.101,Z 99,A -22.6747,B 24.9274,C -1.9681,E1 25.152,E2 467.8888} C_DIS
LIN {X 91.3453,Y -28.0789,Z 99,A -21.3944,B 24.9271,C -1.9724,E1 25.1531,E2 466.6056} C_DIS
LIN {X 92.1041,Y -25.4853,Z 99,A -19.7983,B 24.9268,C -1.9765,E1 25.1543,E2 465.0089} C_DIS
LIN {X 92.9782,Y -22.0844,Z 99,A -17.7063,B 24.9263,C -1.9827,E1 25.1557,E2 462.9144} C_DIS
LIN {X 93.6738,Y -18.9115,Z 99,A -15.7703,B 24.9259,C -1.9885,E1 25.1568,E2 460.9759} C_DIS
LIN {X 94.1597,Y -16.3283,Z 99,A -14.208,B 24.9255,C -1.993,E1 25.1576,E2 459.4122} C_DIS
LIN {X 94.6573,Y -13.1313,Z 99,A -12.2521,B 24.925,C -1.9999,E1 25.1584,E2 457.4515} C_DIS
LIN {X 94.9823,Y -10.5371,Z 99,A -10.7242,B 24.9247,C -2.0034,E1 25.1589,E2 455.9245} C_DIS
LIN {X 95.2118,Y -8.2084,Z 99,A -9.3306,B 24.9244,C -2.0075,E1 25.1593,E2 454.5292} C_DIS
LIN {X 95.3657,Y -6.1489,Z 99,A -8.0651,B 24.924,C -2.0126,E1 25.1595,E2 453.2593} C_DIS
LIN {X 95.5163,Y -2.9933,Z 99,A -6.1347,B 24.9235,C -2.0201,E1 25.1597,E2 451.3226} C_DIS
LIN {X 95.5625,Y -0.3863,Z 99,A -4.5046,B 24.9229,C -2.0278,E1 25.1597,E2 449.6842} C_DIS
LIN {X 95.5134,Y 3.0888,Z 99,A -2.5358,B 24.9227,C -2.03,E1 25.1597,E2 447.7218} C_DIS
LIN {X 95.4007,Y 5.58,Z 99,A -1.0807,B 24.9225,C -2.0332,E1 25.1594,E2 446.2678} C_DIS
LIN {X 95.13,Y 9.0942,Z 99,A 1.0132,B 24.922,C -2.0392,E1 25.159,E2 444.1721} C_DIS
LIN {X 94.7319,Y 12.5814,Z 99,A 3.104,B 24.9216,C -2.0454,E1 25.1582,E2 442.0793} C_DIS
LIN {X 94.3535,Y 15.1679,Z 99,A 4.629,B 24.9213,C -2.0486,E1 25.1576,E2 440.5555} C_DIS
LIN {X 93.7284,Y 18.6454,Z 99,A 6.7348,B 24.9208,C -2.0548,E1 25.1565,E2 438.4475} C_DIS
LIN {X 93.3021,Y 20.6672,Z 99,A 7.9947,B 24.9205,C -2.0595,E1 25.1558,E2 437.1839} C_DIS
LIN {X 92.768,Y 22.9462,Z 99,A 9.5639,B 24.9196,C -2.0702,E1 25.1547,E2 435.5985} C_DIS
LIN {X 91.8573,Y 26.3564,Z 99,A 11.4914,B 24.9196,C -2.0693,E1 25.1533,E2 433.684} C_DIS
LIN {X 90.9451,Y 29.3483,Z 99,A 13.4191,B 24.9191,C -2.077,E1 25.1517,E2 431.7492} C_DIS
LIN {X 89.9743,Y 32.2069,Z 99,A 15.121,B 24.9191,C -2.0782,E1 25.1501,E2 430.0541} C_DIS
LIN {X 89.0609,Y 34.6495,Z 99,A 16.8152,B 24.9183,C -2.0878,E1 25.1484,E2 428.3465} C_DIS
LIN {X 87.9476,Y 37.3851,Z 99,A 18.4365,B 24.9183,C -2.0872,E1 25.1467,E2 426.7356} C_DIS
LIN {X 87.0088,Y 39.5206,Z 99,A 19.858,B 24.9179,C -2.0921,E1 25.1451,E2 425.3103} C_DIS
LIN {X 85.9758,Y 41.7208,Z 99,A 21.2695,B 24.9177,C -2.0944,E1 25.1434,E2 423.9009} C_DIS
LIN {X 84.9529,Y 43.7657,Z 99,A 22.6668,B 24.9174,C -2.0992,E1 25.1416,E2 422.4996} C_DIS
LIN {X 83.7244,Y 46.0748,Z 99,A 24.1972,B 24.9171,C -2.1021,E1 25.1396,E2 420.9706} C_DIS
LIN {X 82.2861,Y 48.5935,Z 99,A 26.0164,B 24.9165,C -2.1098,E1 25.137,E2 419.1425} C_DIS
LIN {X 80.7341,Y 51.1338,Z 99,A 27.6985,B 24.9165,C -2.1105,E1 25.1345,E2 417.4672} C_DIS
LIN {X 78.9581,Y 53.8335,Z 99,A 29.6266,B 24.9161,C -2.1152,E1 25.1315,E2 415.5377} C_DIS
LIN {X 77.6454,Y 55.7098,Z 99,A 31.0016,B 24.9158,C -2.1187,E1 25.1293,E2 414.1611} C_DIS
LIN {X 76.0554,Y 57.8641,Z 99,A 32.5897,B 24.9156,C -2.122,E1 25.1267,E2 412.5729} C_DIS
LIN {X 74.2456,Y 60.1657,Z 99,A 34.4488,B 24.9149,C -2.1301,E1 25.1234,E2 410.7033} C_DIS
LIN {X 71.9796,Y 62.8591,Z 99,A 36.5241,B 24.9146,C -2.1337,E1 25.1196,E2 408.629} C_DIS
LIN {X 69.7263,Y 65.3499,Z 99,A 38.5747,B 24.9141,C -2.1395,E1 25.1158,E2 406.5735} C_DIS
LIN {X 67.52,Y 67.6287,Z 99,A 40.5165,B 24.9137,C -2.1451,E1 25.1119,E2 404.6268} C_DIS
LIN {X 65.0141,Y 70.0414,Z 99,A 42.6133,B 24.9133,C -2.1498,E1 25.1077,E2 402.5275} C_DIS
LIN {X 62.4121,Y 72.3698,Z 99,A 44.704,B 24.913,C -2.1538,E1 25.1033,E2 400.4356} C_DIS
LIN {X 59.8305,Y 74.5173,Z 99,A 46.6837,B 24.9128,C -2.1563,E1 25.099,E2 398.4575} C_DIS
LIN {X 57.1782,Y 76.5706,Z 99,A 48.5334,B 24.913,C -2.154,E1 25.0949,E2 396.62} C_DIS
LIN {X 55.3013,Y 77.9369,Z 99,A 49.9298,B 24.9128,C -2.1565,E1 25.0917,E2 395.2225} C_DIS
LIN {X 52.6265,Y 79.7671,Z 99,A 51.9005,B 24.9124,C -2.1607,E1 25.0872,E2 393.2485} C_DIS
LIN {X 50.3707,Y 81.2109,Z 99,A 53.4258,B 24.9124,C -2.1602,E1 25.0836,E2 391.7293} C_DIS
LIN {X 48.3699,Y 82.4183,Z 99,A 55.0327,B 24.9117,C -2.1698,E1 25.0797,E2 390.1046} C_DIS
LIN {X 45.2848,Y 84.1529,Z 99,A 56.9374,B 24.9121,C -2.1648,E1 25.0751,E2 388.2173} C_DIS
LIN {X 42.9654,Y 85.3619,Z 99,A 58.5006,B 24.912,C -2.1666,E1 25.0712,E2 386.6542} C_DIS
LIN {X 40.1871,Y 86.7026,Z 99,A 60.4095,B 24.9116,C -2.171,E1 25.0663,E2 384.7397} C_DIS
LIN {X 37.6601,Y 87.8316,Z 99,A 62.0016,B 24.9116,C -2.1704,E1 25.0623,E2 383.153} C_DIS
LIN {X 35.4976,Y 88.7276,Z 99,A 63.3992,B 24.9116,C -2.1716,E1 25.0587,E2 381.7557} C_DIS
LIN {X 33.2959,Y 89.5771,Z 99,A 64.8135,B 24.9114,C -2.173,E1 25.055,E2 380.3413} C_DIS
LIN {X 29.9913,Y 90.7368,Z 99,A 67.1277,B 24.9107,C -2.1825,E1 25.0488,E2 378.0091} C_DIS
LIN {X 26.8814,Y 91.7051,Z 99,A 68.8883,B 24.9111,C -2.177,E1 25.0442,E2 376.2644} C_DIS
LIN {X 23.4942,Y 92.6307,Z 99,A 70.9917,B 24.911,C -2.1783,E1 25.0385,E2 374.1613} C_DIS
LIN {X 21.216,Y 93.1789,Z 99,A 72.3981,B 24.911,C -2.1791,E1 25.0347,E2 372.755} C_DIS
LIN {X 17.7623,Y 93.8985,Z 99,A 74.5071,B 24.9109,C -2.1798,E1 25.0289,E2 370.6469} C_DIS
LIN {X 15.1862,Y 94.3507,Z 99,A 76.0446,B 24.9109,C -2.1793,E1 25.0247,E2 369.1123} C_DIS
LIN {X 11.71,Y 94.8448,Z 99,A 78.1495,B 24.9109,C -2.1798,E1 25.0188,E2 367.008} C_DIS
LIN {X 9.6975,Y 95.0702,Z 99,A 79.4045,B 24.9107,C -2.1814,E1 25.0153,E2 365.7499} C_DIS
LIN {X 7.0317,Y 95.306,Z 99,A 80.9674,B 24.9109,C -2.18,E1 25.011,E2 364.1912} C_DIS
LIN {X 4.6957,Y 95.4495,Z 99,A 82.3701,B 24.9109,C -2.18,E1 25.0071,E2 362.7891} C_DIS
LIN {X 2.3571,Y 95.5359,Z 99,A 83.7726,B 24.9109,C -2.1798,E1 25.0032,E2 361.3873} C_DIS
LIN {X 0.0046,Y 95.565,Z 99,A 85.1848,B 24.9109,C -2.1796,E1 24.9992,E2 359.9756} C_DIS
LIN {X -3.5194,Y 95.5002,Z 99,A 87.5039,B 24.9104,C -2.1862,E1 24.9927,E2 357.6407} C_DIS
LIN {X -7.0221,Y 95.3066,Z 99,A 89.4039,B 24.911,C -2.1783,E1 24.9875,E2 355.7587} C_DIS
LIN {X -10.5145,Y 94.9847,Z 99,A 91.5106,B 24.911,C -2.1774,E1 24.9816,E2 353.6531} C_DIS
LIN {X -13.4201,Y 94.6162,Z 99,A 93.3838,B 24.9108,C -2.1803,E1 24.9764,E2 351.7714} C_DIS
LIN {X -17.2155,Y 94.0003,Z 99,A 95.6075,B 24.9112,C -2.1758,E1 24.9703,E2 349.5562} C_DIS
LIN {X -19.7814,Y 93.4952,Z 99,A 97.2674,B 24.9111,C -2.1777,E1 24.9658,E2 347.8901} C_DIS
LIN {X -22.7003,Y 92.828,Z 99,A 99.041,B 24.9112,C -2.1753,E1 24.9609,E2 346.1197} C_DIS
LIN {X -25.4873,Y 92.1036,Z 99,A 100.678,B 24.9116,C -2.1704,E1 24.9566,E2 344.4917} C_DIS
LIN {X -27.7759,Y 91.4392,Z 99,A 102.3094,B 24.9112,C -2.1757,E1 24.9522,E2 342.845} C_DIS
LIN {X -30.7876,Y 90.4684,Z 99,A 104.1332,B 24.9116,C -2.171,E1 24.9473,E2 341.0291} C_DIS
LIN {X -33.9685,Y 89.3224,Z 99,A 106.1158,B 24.9119,C -2.1669,E1 24.9422,E2 339.0523} C_DIS
LIN {X -37.3858,Y 87.9472,Z 99,A 108.2601,B 24.9124,C -2.1616,E1 24.9366,E2 336.9157} C_DIS
LIN {X -39.4165,Y 87.0557,Z 99,A 109.6516,B 24.9124,C -2.1617,E1 24.9331,E2 335.5206} C_DIS
LIN {X -41.8748,Y 85.9018,Z 99,A 111.2207,B 24.9127,C -2.1572,E1 24.9292,E2 333.9582} C_DIS
LIN {X -44.5861,Y 84.5246,Z 99,A 113.1481,B 24.9127,C -2.1577,E1 24.9244,E2 332.0245} C_DIS
LIN {X -46.8584,Y 83.2869,Z 99,A 114.6519,B 24.913,C -2.1534,E1 24.9207,E2 330.5265} C_DIS
LIN {X -49.1368,Y 81.9649,Z 99,A 116.2002,B 24.9133,C -2.1495,E1 24.917,E2 328.9828} C_DIS
LIN {X -51.1286,Y 80.7375,Z 99,A 117.6094,B 24.9135,C -2.1471,E1 24.9136,E2 327.5749} C_DIS
LIN {X -53.8313,Y 78.9596,Z 99,A 119.558,B 24.9138,C -2.1436,E1 24.9091,E2 325.6281} C_DIS
LIN {X -55.9713,Y 77.4589,Z 99,A 121.1325,B 24.9141,C -2.1407,E1 24.9055,E2 324.0551} C_DIS
LIN {X -58.3161,Y 75.7071,Z 99,A 123.0115,B 24.9141,C -2.1411,E1 24.9013,E2 322.1684} C_DIS
LIN {X -61.0747,Y 73.4998,Z 99,A 125.1322,B 24.9144,C -2.1366,E1 24.8968,E2 320.0505} C_DIS
LIN {X -63.7295,Y 71.2101,Z 99,A 127.2465,B 24.9147,C -2.1322,E1 24.8923,E2 317.9382} C_DIS
LIN {X -66.2967,Y 68.8264,Z 99,A 129.369,B 24.9151,C -2.128,E1 24.888,E2 315.817} C_DIS
LIN {X -68.8046,Y 66.3194,Z 99,A 131.4934,B 24.9155,C -2.1228,E1 24.8839,E2 313.696} C_DIS
LIN {X -71.1894,Y 63.7526,Z 99,A 133.6078,B 24.9159,C -2.118,E1 24.8799,E2 311.5837} C_DIS
LIN {X -73.3878,Y 61.2094,Z 99,A 135.663,B 24.9162,C -2.1141,E1 24.8762,E2 309.5284} C_DIS
LIN {X -75.6124,Y 58.4389,Z 99,A 137.7781,B 24.9167,C -2.1079,E1 24.8725,E2 307.418} C_DIS
LIN {X -77.4085,Y 56.0403,Z 99,A 139.4656,B 24.9173,C -2.0995,E1 24.8698,E2 305.7423} C_DIS
LIN {X -78.791,Y 54.0798,Z 99,A 140.922,B 24.9176,C -2.0962,E1 24.8674,E2 304.2869} C_DIS
LIN {X -80.0891,Y 52.1381,Z 99,A 142.3259,B 24.9179,C -2.0924,E1 24.8653,E2 302.8849} C_DIS
LIN {X -81.8256,Y 49.3659,Z 99,A 144.3042,B 24.9183,C -2.0874,E1 24.8624,E2 300.9084} C_DIS
LIN {X -83.0101,Y 47.3472,Z 99,A 145.7462,B 24.9185,C -2.0846,E1 24.8604,E2 299.4656} C_DIS
LIN {X -84.1446,Y 45.3001,Z 99,A 147.159,B 24.9188,C -2.0808,E1 24.8585,E2 298.0544} C_DIS
LIN {X -85.5686,Y 42.5483,Z 99,A 149.1044,B 24.919,C -2.0781,E1 24.856,E2 296.105} C_DIS
LIN {X -86.779,Y 40.023,Z 99,A 150.7238,B 24.9196,C -2.0712,E1 24.8541,E2 294.4933} C_DIS
LIN {X -87.841,Y 37.638,Z 99,A 152.2628,B 24.92,C -2.0656,E1 24.8524,E2 292.9591} C_DIS
LIN {X -88.7355,Y 35.4778,Z 99,A 153.6719,B 24.9203,C -2.0615,E1 24.8509,E2 291.5519} C_DIS
LIN {X -89.577,Y 33.2961,Z 99,A 155.0873,B 24.9206,C -2.0576,E1 24.8495,E2 290.1378} C_DIS
LIN {X -90.7385,Y 29.9865,Z 99,A 157.3884,B 24.9206,C -2.0574,E1 24.8474,E2 287.8241} C_DIS
LIN {X -91.7047,Y 26.8826,Z 99,A 159.1964,B 24.9214,C -2.0468,E1 24.846,E2 286.0309} C_DIS
LIN {X -92.6277,Y 23.5057,Z 99,A 161.3177,B 24.9219,C -2.0409,E1 24.8444,E2 283.9114} C_DIS
LIN {X -93.1674,Y 21.2654,Z 99,A 162.7129,B 24.9222,C -2.037,E1 24.8436,E2 282.5174} C_DIS
LIN {X -93.8927,Y 17.7923,Z 99,A 164.8459,B 24.9227,C -2.0304,E1 24.8424,E2 280.3875} C_DIS
LIN {X -94.3419,Y 15.2385,Z 99,A 166.3699,B 24.9232,C -2.0244,E1 24.8417,E2 278.8687} C_DIS
LIN {X -94.7979,Y 12.072,Z 99,A 168.3631,B 24.9234,C -2.0207,E1 24.8409,E2 276.8726} C_DIS
LIN {X -95.0758,Y 9.6441,Z 99,A 169.8227,B 24.9238,C -2.0158,E1 24.8405,E2 275.4159} C_DIS
LIN {X -95.3066,Y 7.0232,Z 99,A 171.3727,B 24.9243,C -2.0098,E1 24.8401,E2 273.8709} C_DIS
LIN {X -95.4493,Y 4.6995,Z 99,A 172.7808,B 24.9246,C -2.0057,E1 24.8399,E2 272.464} C_DIS
LIN {X -95.5362,Y 2.3467,Z 99,A 174.2039,B 24.9249,C -2.0015,E1 24.8399,E2 271.0424} C_DIS
LIN {X -95.5646,Y 0.0051,Z 99,A 175.8042,B 24.9248,C -2.0033,E1 24.8398,E2 269.4283} C_DIS
LIN {X -95.5084,Y -3.2508,Z 99,A 177.6147,B 24.9256,C -1.9925,E1 24.8399,E2 267.6325} C_DIS
LIN {X -95.4001,Y -5.5895,Z 99,A 179.0272,B 24.9259,C -1.9883,E1 24.8401,E2 266.2216} C_DIS
LIN {X -95.1303,Y -9.0911,Z 99,A -178.8526,B 24.9263,C -1.9821,E1 24.8406,E2 264.1035} C_DIS
LIN {X -94.7679,Y -12.3034,Z 99,A -176.8256,B 24.9266,C -1.9788,E1 24.8413,E2 262.0722} C_DIS
LIN {X -94.3509,Y -15.1848,Z 99,A -175.1742,B 24.9272,C -1.9703,E1 24.842,E2 260.4313} C_DIS
LIN {X -93.7292,Y -18.6414,Z 99,A -173.052,B 24.9277,C -1.9642,E1 24.8431,E2 258.311} C_DIS
LIN {X -93.3029,Y -20.6637,Z 99,A -171.7838,B 24.9279,C -1.9613,E1 24.8438,E2 257.0422} C_DIS
LIN {X -92.7602,Y -22.9781,Z 99,A -170.336,B 24.9281,C -1.9577,E1 24.8448,E2 255.5946} C_DIS
LIN {X -92.1003,Y -25.4991,Z 99,A -168.8025,B 24.9286,C -1.952,E1 24.8459,E2 254.0659} C_DIS
LIN {X -91.4502,Y -27.7406,Z 99,A -167.3877,B 24.9288,C -1.9482,E1 24.847,E2 252.6518} C_DIS
LIN {X -90.4603,Y -30.8116,Z 99,A -165.4073,B 24.9291,C -1.944,E1 24.8488,E2 250.6702} C_DIS
LIN {X -89.5772,Y -33.2956,Z 99,A -163.8496,B 24.9295,C -1.9386,E1 24.8502,E2 249.1166} C_DIS
LIN {X -88.7351,Y -35.4789,Z 99,A -162.4376,B 24.9298,C -1.9348,E1 24.8517,E2 247.7058} C_DIS
LIN {X -87.6035,Y -38.1831,Z 99,A -160.5981,B 24.93,C -1.9324,E1 24.8537,E2 245.8617} C_DIS
LIN {X -86.3896,Y -40.8597,Z 99,A -158.8958,B 24.9305,C -1.9255,E1 24.8557,E2 244.1667} C_DIS
LIN {X -85.3626,Y -42.9639,Z 99,A -157.2595,B 24.9302,C -1.9291,E1 24.8577,E2 242.5128} C_DIS
LIN {X -83.7181,Y -46.0863,Z 99,A -155.3589,B 24.9312,C -1.9163,E1 24.8602,E2 240.6327} C_DIS
LIN {X -82.572,Y -48.1094,Z 99,A -153.9557,B 24.9314,C -1.9129,E1 24.8622,E2 239.2303} C_DIS
LIN {X -80.7636,Y -51.0868,Z 99,A -151.6857,B 24.9314,C -1.9134,E1 24.8655,E2 236.9477} C_DIS
LIN {X -79.0283,Y -53.7298,Z 99,A -149.7661,B 24.9317,C -1.9093,E1 24.8685,E2 235.028} C_DIS
LIN {X -77.0424,Y -56.5403,Z 99,A -147.7876,B 24.9322,C -1.9014,E1 24.8717,E2 233.0588} C_DIS
LIN {X -75.3344,Y -58.7996,Z 99,A -145.9486,B 24.9322,C -1.902,E1 24.8749,E2 231.2098} C_DIS
LIN {X -73.1265,Y -61.5238,Z 99,A -143.8348,B 24.9325,C -1.8974,E1 24.8786,E2 229.097} C_DIS
LIN {X -70.8206,Y -64.1646,Z 99,A -141.7172,B 24.9328,C -1.8932,E1 24.8826,E2 226.98} C_DIS
LIN {X -67.9952,Y -67.149,Z 99,A -139.3724,B 24.9335,C -1.884,E1 24.8871,E2 224.6471} C_DIS
LIN {X -65.6036,Y -69.4876,Z 99,A -137.3703,B 24.9338,C -1.8797,E1 24.8911,E2 222.6468} C_DIS
LIN {X -63.304,Y -71.591,Z 99,A -135.3543,B 24.9337,C -1.8809,E1 24.8953,E2 220.6199} C_DIS
LIN {X -60.6365,Y -73.8639,Z 99,A -133.2466,B 24.9339,C -1.8772,E1 24.8999,E2 218.513} C_DIS
LIN {X -57.8891,Y -76.0361,Z 99,A -131.2281,B 24.9344,C -1.8707,E1 24.9043,E2 216.5026} C_DIS
Enddeposition()
END
